LIN {X 0,Y 473.867,Z 372.012,A -85,B 0,C 180,E1 -7419.027,E2 -7419.027} C_VEL
LIN {X 0,Y 473.751,Z 376.078,A -85,B 0,C 180,E1 -7420.747,E2 -7420.747} C_VEL
LIN {X 0,Y 473.643,Z 378.041,A -85,B 0,C 180,E1 -7422.107,E2 -7422.107} C_VEL
LIN {X 0,Y 473.594,Z 378.94,A -85,B 0,C 180,E1 -7423.354,E2 -7423.354} C_VEL
LIN {X 0,Y 473.663,Z 378.958,A -85,B 0,C 180,E1 -7424.587,E2 -7424.587} C_VEL
LIN {X 0,Y 473.668,Z 378.173,A -85,B 0,C 180,E1 -7425.786,E2 -7425.786} C_VEL
LIN {X 0,Y 473.687,Z 376.639,A -85,B 0,C 180,E1 -7426.962,E2 -7426.962} C_VEL
LIN {X 0,Y 473.768,Z 374.355,A -85,B 0,C 180,E1 -7428.123,E2 -7428.123} C_VEL
LIN {X 0,Y 473.919,Z 369.986,A -85,B 0,C 180,E1 -7429.66,E2 -7429.66} C_VEL
LIN {X 0,Y 474.11,Z 365.022,A -85,B 0,C 180,E1 -7430.975,E2 -7430.975} C_VEL
LIN {X 0,Y 474.333,Z 358.198,A -85,B 0,C 180,E1 -7432.389,E2 -7432.389} C_VEL
LIN {X 0,Y 474.456,Z 355.246,A -85,B 0,C 180,E1 -7432.903,E2 -7432.903} C_VEL
LIN {X 0,Y 473.946,Z 351.766,A -85,B 0,C 180,E1 -7433.474,E2 -7433.474} C_VEL
LIN {X 0,Y 471.408,Z 345.796,A -85,B 0,C 180,E1 -7434.387,E2 -7434.387} C_VEL
LIN {X 0,Y 468.889,Z 339.334,A -85,B 0,C 180,E1 -7435.251,E2 -7435.251} C_VEL
LIN {X 0,Y 468.41,Z 335.005,A -85,B 0,C 180,E1 -7435.739,E2 -7435.739} C_VEL
LIN {X 0,Y 468.871,Z 324.63,A -85,B 0,C 180,E1 -7436.713,E2 -7436.713} C_VEL
LIN {X 0,Y 469.311,Z 314.156,A -85,B 0,C 180,E1 -7437.505,E2 -7437.505} C_VEL
LIN {X 0,Y 469.802,Z 301.748,A -85,B 0,C 180,E1 -7438.239,E2 -7438.239} C_VEL
LIN {X 0,Y 470.133,Z 288.339,A -85,B 0,C 180,E1 -7438.813,E2 -7438.813} C_VEL
LIN {X 0,Y 470.416,Z 274.959,A -85,B 0,C 180,E1 -7439.193,E2 -7439.193} C_VEL
LIN {X 0,Y 471.25,Z 183.279,A -85,B 0,C 180,E1 -7440.659,E2 -7440.659} C_VEL
LIN {X 0,Y 468.411,Z 168.295,A -85,B 0,C 180,E1 -7441.031,E2 -7441.031} C_VEL
LIN {X 0,Y 468.965,Z 153.603,A -85,B 0,C 180,E1 -7444.048,E2 -7444.048} C_VEL
LIN {X 0,Y 467.574,Z 145.244,A -85,B 0,C 180,E1 -7445.881,E2 -7445.881} C_VEL
LIN {X 0,Y 467.606,Z 145.236,A -85,B 0,C 180,E1 -7449.777,E2 -7449.777} C_VEL
LIN {X 0,Y 467.56,Z 145.247,A -85,B 0,C 180,E1 -7452.505,E2 -7452.505} C_VEL
LIN {X 0,Y 467.586,Z 145.236,A -85,B 0,C 180,E1 -7455.196,E2 -7455.196} C_VEL
LIN {X 0,Y 467.644,Z 145.231,A -85,B 0,C 180,E1 -7457.855,E2 -7457.855} C_VEL
LIN {X 0,Y 467.629,Z 145.231,A -85,B 0,C 180,E1 -7461.357,E2 -7461.357} C_VEL
LIN {X 0,Y 467.696,Z 145.227,A -85,B 0,C 180,E1 -7463.962,E2 -7463.962} C_VEL
LIN {X 0,Y 467.808,Z 145.209,A -85,B 0,C 180,E1 -7467.417,E2 -7467.417} C_VEL
LIN {X 0,Y 467.845,Z 145.211,A -85,B 0,C 180,E1 -7470,E2 -7470} C_VEL
LIN {X 0,Y 467.808,Z 145.21,A -85,B 0,C 180,E1 -7472.583,E2 -7472.583} C_VEL
LIN {X 0,Y 467.696,Z 145.229,A -85,B 0,C 180,E1 -7476.038,E2 -7476.038} C_VEL
LIN {X 0,Y 467.629,Z 145.231,A -85,B 0,C 180,E1 -7478.644,E2 -7478.644} C_VEL
LIN {X 0,Y 467.644,Z 145.232,A -85,B 0,C 180,E1 -7482.146,E2 -7482.146} C_VEL
LIN {X 0,Y 467.609,Z 145.241,A -85,B 0,C 180,E1 -7485.696,E2 -7485.696} C_VEL
LIN {X 0,Y 467.568,Z 145.238,A -85,B 0,C 180,E1 -7488.748,E2 -7488.748} C_VEL
LIN {X 0,Y 467.554,Z 145.243,A -85,B 0,C 180,E1 -7491.261,E2 -7491.261} C_VEL
LIN {X 0,Y 467.546,Z 145.244,A -85,B 0,C 180,E1 -7493.944,E2 -7493.944} C_VEL
LIN {X 0,Y 467.53,Z 145.244,A -85,B 0,C 180,E1 -7496.805,E2 -7496.805} C_VEL
LIN {X 0,Y 467.509,Z 145.249,A -85,B 0,C 180,E1 -7499.741,E2 -7499.741} C_VEL
LIN {X 0,Y 467.568,Z 145.239,A -85,B 0,C 180,E1 -7502.759,E2 -7502.759} C_VEL
LIN {X 0,Y 467.544,Z 145.242,A -85,B 0,C 180,E1 -7505.89,E2 -7505.89} C_VEL
LIN {X 0,Y 467.539,Z 145.249,A -85,B 0,C 180,E1 -7509.148,E2 -7509.148} C_VEL
LIN {X 0,Y 467.552,Z 145.245,A -85,B 0,C 180,E1 -7511.405,E2 -7511.405} C_VEL
LIN {X 0,Y 467.56,Z 145.247,A -85,B 0,C 180,E1 -7515.052,E2 -7515.052} C_VEL
LIN {X 0,Y 467.554,Z 145.244,A -85,B 0,C 180,E1 -7518.726,E2 -7518.726} C_VEL
LIN {X 0,Y 467.534,Z 145.242,A -85,B 0,C 180,E1 -7521.953,E2 -7521.953} C_VEL
LIN {X 0,Y 467.544,Z 145.245,A -85,B 0,C 180,E1 -7525.166,E2 -7525.166} C_VEL
LIN {X 0,Y 467.55,Z 145.242,A -85,B 0,C 180,E1 -7528.258,E2 -7528.258} C_VEL
LIN {X 0,Y 467.532,Z 145.244,A -85,B 0,C 180,E1 -7531.248,E2 -7531.248} C_VEL
LIN {X 0,Y 467.571,Z 145.243,A -85,B 0,C 180,E1 -7534.401,E2 -7534.401} C_VEL
LIN {X 0,Y 467.544,Z 145.244,A -85,B 0,C 180,E1 -7536.995,E2 -7536.995} C_VEL
LIN {X 0,Y 467.6,Z 145.235,A -85,B 0,C 180,E1 -7539.777,E2 -7539.777} C_VEL
LIN {X 0,Y 467.558,Z 145.247,A -85,B 0,C 180,E1 -7542.505,E2 -7542.505} C_VEL
LIN {X 0,Y 467.584,Z 145.237,A -85,B 0,C 180,E1 -7545.196,E2 -7545.196} C_VEL
LIN {X 0,Y 467.641,Z 145.231,A -85,B 0,C 180,E1 -7547.855,E2 -7547.855} C_VEL
LIN {X 0,Y 467.623,Z 145.231,A -85,B 0,C 180,E1 -7551.357,E2 -7551.357} C_VEL
LIN {X 0,Y 467.693,Z 145.227,A -85,B 0,C 180,E1 -7553.962,E2 -7553.962} C_VEL
LIN {X 0,Y 467.805,Z 145.209,A -85,B 0,C 180,E1 -7557.417,E2 -7557.417} C_VEL
LIN {X 0,Y 467.842,Z 145.211,A -85,B 0,C 180,E1 -7560,E2 -7560} C_VEL
LIN {X 0,Y 467.805,Z 145.21,A -85,B 0,C 180,E1 -7562.584,E2 -7562.584} C_VEL
LIN {X 0,Y 467.693,Z 145.229,A -85,B 0,C 180,E1 -7566.038,E2 -7566.038} C_VEL
LIN {X 0,Y 467.627,Z 145.231,A -85,B 0,C 180,E1 -7568.644,E2 -7568.644} C_VEL
LIN {X 0,Y 467.642,Z 145.232,A -85,B 0,C 180,E1 -7572.146,E2 -7572.146} C_VEL
LIN {X 0,Y 467.607,Z 145.241,A -85,B 0,C 180,E1 -7575.696,E2 -7575.696} C_VEL
LIN {X 0,Y 467.567,Z 145.238,A -85,B 0,C 180,E1 -7578.748,E2 -7578.748} C_VEL
LIN {X 0,Y 467.553,Z 145.244,A -85,B 0,C 180,E1 -7581.261,E2 -7581.261} C_VEL
LIN {X 0,Y 467.546,Z 145.244,A -85,B 0,C 180,E1 -7583.945,E2 -7583.945} C_VEL
LIN {X 0,Y 467.53,Z 145.244,A -85,B 0,C 180,E1 -7586.806,E2 -7586.806} C_VEL
LIN {X 0,Y 467.505,Z 145.249,A -85,B 0,C 180,E1 -7589.742,E2 -7589.742} C_VEL
LIN {X 0,Y 467.569,Z 145.24,A -85,B 0,C 180,E1 -7592.76,E2 -7592.76} C_VEL
LIN {X 0,Y 467.54,Z 145.243,A -85,B 0,C 180,E1 -7595.891,E2 -7595.891} C_VEL
LIN {X 0,Y 467.54,Z 145.25,A -85,B 0,C 180,E1 -7599.149,E2 -7599.149} C_VEL
LIN {X 0,Y 467.556,Z 145.244,A -85,B 0,C 180,E1 -7601.406,E2 -7601.406} C_VEL
LIN {X 0,Y 467.56,Z 145.247,A -85,B 0,C 180,E1 -7605.052,E2 -7605.052} C_VEL
LIN {X 0,Y 467.559,Z 145.244,A -85,B 0,C 180,E1 -7608.726,E2 -7608.726} C_VEL
LIN {X 0,Y 467.539,Z 145.242,A -85,B 0,C 180,E1 -7611.953,E2 -7611.953} C_VEL
LIN {X 0,Y 467.549,Z 145.244,A -85,B 0,C 180,E1 -7615.166,E2 -7615.166} C_VEL
LIN {X 0,Y 467.546,Z 145.243,A -85,B 0,C 180,E1 -7618.257,E2 -7618.257} C_VEL
LIN {X 0,Y 467.524,Z 145.247,A -85,B 0,C 180,E1 -7621.247,E2 -7621.247} C_VEL
LIN {X 0,Y 467.556,Z 145.305,A -85,B 0,C 180,E1 -7624.376,E2 -7624.376} C_VEL
LIN {X 0,Y 469.555,Z 155.653,A -85,B 0,C 180,E1 -7626.398,E2 -7626.398} C_VEL
LIN {X 0,Y 469.662,Z 160.735,A -85,B 0,C 180,E1 -7627.336,E2 -7627.336} C_VEL
LIN {X 0,Y 468.796,Z 180.844,A -85,B 0,C 180,E1 -7630.944,E2 -7630.944} C_VEL
LIN {X 0,Y 468.312,Z 192.554,A -85,B 0,C 180,E1 -7633.016,E2 -7633.016} C_VEL
LIN {X 0,Y 471.118,Z 211.466,A -85,B 0,C 180,E1 -7633.427,E2 -7633.427} C_VEL
LIN {X 0,Y 470.386,Z 301.176,A -85,B 0,C 180,E1 -7634.871,E2 -7634.871} C_VEL
LIN {X 0,Y 470.014,Z 314.178,A -85,B 0,C 180,E1 -7635.246,E2 -7635.246} C_VEL
LIN {X 0,Y 469.599,Z 326.238,A -85,B 0,C 180,E1 -7635.759,E2 -7635.759} C_VEL
LIN {X 0,Y 469.091,Z 338.452,A -85,B 0,C 180,E1 -7636.462,E2 -7636.462} C_VEL
LIN {X 0,Y 468.604,Z 349.481,A -85,B 0,C 180,E1 -7637.282,E2 -7637.282} C_VEL
LIN {X 0,Y 468.158,Z 360.491,A -85,B 0,C 180,E1 -7638.307,E2 -7638.307} C_VEL
LIN {X 0,Y 467.699,Z 369.878,A -85,B 0,C 180,E1 -7639.393,E2 -7639.393} C_VEL
LIN {X 0,Y 467.276,Z 378.958,A -85,B 0,C 180,E1 -7640.695,E2 -7640.695} C_VEL
LIN {X 0,Y 467.007,Z 386.273,A -85,B 0,C 180,E1 -7641.998,E2 -7641.998} C_VEL
LIN {X 0,Y 466.842,Z 391.213,A -85,B 0,C 180,E1 -7643.083,E2 -7643.083} C_VEL
LIN {X 0,Y 466.756,Z 396.008,A -85,B 0,C 180,E1 -7644.383,E2 -7644.383} C_VEL
LIN {X 0,Y 466.645,Z 399.671,A -85,B 0,C 180,E1 -7645.681,E2 -7645.681} C_VEL
LIN {X 0,Y 466.689,Z 401.563,A -85,B 0,C 180,E1 -7646.546,E2 -7646.546} C_VEL
LIN {X 0,Y 466.662,Z 402.984,A -85,B 0,C 180,E1 -7647.41,E2 -7647.41} C_VEL
LIN {X 0,Y 466.62,Z 404.604,A -85,B 0,C 180,E1 -7649.137,E2 -7649.137} C_VEL
LIN {X 0,Y 466.602,Z 404.824,A -85,B 0,C 180,E1 -7650,E2 -7650} C_VEL
LIN {X 0,Y 466.62,Z 404.606,A -85,B 0,C 180,E1 -7650.863,E2 -7650.863} C_VEL
LIN {X 0,Y 466.662,Z 402.978,A -85,B 0,C 180,E1 -7652.589,E2 -7652.589} C_VEL
LIN {X 0,Y 466.688,Z 401.562,A -85,B 0,C 180,E1 -7653.453,E2 -7653.453} C_VEL
LIN {X 0,Y 466.687,Z 398.586,A -85,B 0,C 180,E1 -7654.751,E2 -7654.751} C_VEL
LIN {X 0,Y 466.743,Z 394.561,A -85,B 0,C 180,E1 -7656.05,E2 -7656.05} C_VEL
LIN {X 0,Y 466.94,Z 388.369,A -85,B 0,C 180,E1 -7657.567,E2 -7657.567} C_VEL
LIN {X 0,Y 467.196,Z 381.607,A -85,B 0,C 180,E1 -7658.87,E2 -7658.87} C_VEL
LIN {X 0,Y 467.524,Z 373.225,A -85,B 0,C 180,E1 -7660.173,E2 -7660.173} C_VEL
LIN {X 0,Y 467.975,Z 364.611,A -85,B 0,C 180,E1 -7661.258,E2 -7661.258} C_VEL
LIN {X 0,Y 468.453,Z 354.527,A -85,B 0,C 180,E1 -7662.294,E2 -7662.294} C_VEL
LIN {X 0,Y 468.873,Z 343.464,A -85,B 0,C 180,E1 -7663.213,E2 -7663.213} C_VEL
LIN {X 0,Y 469.446,Z 331.882,A -85,B 0,C 180,E1 -7663.969,E2 -7663.969} C_VEL
LIN {X 0,Y 469.855,Z 319.883,A -85,B 0,C 180,E1 -7664.565,E2 -7664.565} C_VEL
LIN {X 0,Y 470.286,Z 306.964,A -85,B 0,C 180,E1 -7665.021,E2 -7665.021} C_VEL
LIN {X 0,Y 470.57,Z 293.349,A -85,B 0,C 180,E1 -7665.317,E2 -7665.317} C_VEL
LIN {X 0,Y 471.196,Z 210.389,A -85,B 0,C 180,E1 -7666.646,E2 -7666.646} C_VEL
LIN {X 0,Y 468.312,Z 191.835,A -85,B 0,C 180,E1 -7667.087,E2 -7667.087} C_VEL
LIN {X 0,Y 469.027,Z 174.329,A -85,B 0,C 180,E1 -7670.159,E2 -7670.159} C_VEL
LIN {X 0,Y 469.706,Z 157.643,A -85,B 0,C 180,E1 -7673.126,E2 -7673.126} C_VEL
LIN {X 0,Y 469.008,Z 152.49,A -85,B 0,C 180,E1 -7674.099,E2 -7674.099} C_VEL
LIN {X 0,Y 467.555,Z 145.247,A -85,B 0,C 180,E1 -7675.543,E2 -7675.543} C_VEL
LIN {X 0,Y 467.523,Z 145.251,A -85,B 0,C 180,E1 -7678.753,E2 -7678.753} C_VEL
LIN {X 0,Y 467.545,Z 145.249,A -85,B 0,C 180,E1 -7681.742,E2 -7681.742} C_VEL
LIN {X 0,Y 467.548,Z 145.246,A -85,B 0,C 180,E1 -7684.833,E2 -7684.833} C_VEL
LIN {X 0,Y 467.537,Z 145.245,A -85,B 0,C 180,E1 -7688.046,E2 -7688.046} C_VEL
LIN {X 0,Y 467.557,Z 145.248,A -85,B 0,C 180,E1 -7691.273,E2 -7691.273} C_VEL
LIN {X 0,Y 467.56,Z 145.246,A -85,B 0,C 180,E1 -7694.947,E2 -7694.947} C_VEL
LIN {X 0,Y 467.554,Z 145.244,A -85,B 0,C 180,E1 -7698.594,E2 -7698.594} C_VEL
LIN {X 0,Y 467.536,Z 145.245,A -85,B 0,C 180,E1 -7701.412,E2 -7701.412} C_VEL
LIN {X 0,Y 467.545,Z 145.242,A -85,B 0,C 180,E1 -7704.262,E2 -7704.262} C_VEL
LIN {X 0,Y 467.566,Z 145.239,A -85,B 0,C 180,E1 -7707.322,E2 -7707.322} C_VEL
LIN {X 0,Y 467.52,Z 145.248,A -85,B 0,C 180,E1 -7710.677,E2 -7710.677} C_VEL
LIN {X 0,Y 467.528,Z 145.241,A -85,B 0,C 180,E1 -7713.194,E2 -7713.194} C_VEL
LIN {X 0,Y 467.544,Z 145.245,A -85,B 0,C 180,E1 -7716.055,E2 -7716.055} C_VEL
LIN {X 0,Y 467.579,Z 145.239,A -85,B 0,C 180,E1 -7719.775,E2 -7719.775} C_VEL
LIN {X 0,Y 467.55,Z 145.247,A -85,B 0,C 180,E1 -7722.504,E2 -7722.504} C_VEL
LIN {X 0,Y 467.58,Z 145.235,A -85,B 0,C 180,E1 -7725.195,E2 -7725.195} C_VEL
LIN {X 0,Y 467.64,Z 145.233,A -85,B 0,C 180,E1 -7727.854,E2 -7727.854} C_VEL
LIN {X 0,Y 467.625,Z 145.231,A -85,B 0,C 180,E1 -7731.356,E2 -7731.356} C_VEL
LIN {X 0,Y 467.691,Z 145.231,A -85,B 0,C 180,E1 -7733.962,E2 -7733.962} C_VEL
LIN {X 0,Y 467.803,Z 145.212,A -85,B 0,C 180,E1 -7737.416,E2 -7737.416} C_VEL
LIN {X 0,Y 467.84,Z 145.211,A -85,B 0,C 180,E1 -7740,E2 -7740} C_VEL
LIN {X 0,Y 467.803,Z 145.211,A -85,B 0,C 180,E1 -7742.583,E2 -7742.583} C_VEL
LIN {X 0,Y 467.691,Z 145.23,A -85,B 0,C 180,E1 -7746.038,E2 -7746.038} C_VEL
LIN {X 0,Y 467.624,Z 145.234,A -85,B 0,C 180,E1 -7748.643,E2 -7748.643} C_VEL
LIN {X 0,Y 467.639,Z 145.237,A -85,B 0,C 180,E1 -7752.145,E2 -7752.145} C_VEL
LIN {X 0,Y 467.603,Z 145.244,A -85,B 0,C 180,E1 -7755.696,E2 -7755.696} C_VEL
LIN {X 0,Y 467.607,Z 145.241,A -85,B 0,C 180,E1 -7759.308,E2 -7759.308} C_VEL
LIN {X 0,Y 467.602,Z 145.344,A -85,B 0,C 180,E1 -7762.361,E2 -7762.361} C_VEL
LIN {X 0,Y 468.924,Z 152.789,A -85,B 0,C 180,E1 -7763.905,E2 -7763.905} C_VEL
LIN {X 0,Y 468.551,Z 168.51,A -85,B 0,C 180,E1 -7766.983,E2 -7766.983} C_VEL
LIN {X 0,Y 471.425,Z 184.218,A -85,B 0,C 180,E1 -7767.375,E2 -7767.375} C_VEL
LIN {X 0,Y 470.514,Z 276.407,A -85,B 0,C 180,E1 -7768.873,E2 -7768.873} C_VEL
LIN {X 0,Y 470.217,Z 289.972,A -85,B 0,C 180,E1 -7769.276,E2 -7769.276} C_VEL
LIN {X 0,Y 469.877,Z 302.576,A -85,B 0,C 180,E1 -7769.831,E2 -7769.831} C_VEL
LIN {X 0,Y 469.456,Z 313.602,A -85,B 0,C 180,E1 -7770.482,E2 -7770.482} C_VEL
LIN {X 0,Y 468.956,Z 324.82,A -85,B 0,C 180,E1 -7771.327,E2 -7771.327} C_VEL
LIN {X 0,Y 468.447,Z 335.259,A -85,B 0,C 180,E1 -7772.308,E2 -7772.308} C_VEL
LIN {X 0,Y 468.084,Z 344.387,A -85,B 0,C 180,E1 -7773.368,E2 -7773.368} C_VEL
LIN {X 0,Y 467.588,Z 353.449,A -85,B 0,C 180,E1 -7774.672,E2 -7774.672} C_VEL
LIN {X 0,Y 467.28,Z 360.415,A -85,B 0,C 180,E1 -7775.913,E2 -7775.913} C_VEL
LIN {X 0,Y 467.005,Z 365.825,A -85,B 0,C 180,E1 -7777.1,E2 -7777.1} C_VEL
LIN {X 0,Y 466.871,Z 370.84,A -85,B 0,C 180,E1 -7778.486,E2 -7778.486} C_VEL
LIN {X 0,Y 466.709,Z 374.498,A -85,B 0,C 180,E1 -7779.828,E2 -7779.828} C_VEL
LIN {X 0,Y 466.594,Z 377.553,A -85,B 0,C 180,E1 -7781.509,E2 -7781.509} C_VEL
LIN {X 0,Y 466.519,Z 378.782,A -85,B 0,C 180,E1 -7782.68,E2 -7782.68} C_VEL
LIN {X 0,Y 466.527,Z 379.234,A -85,B 0,C 180,E1 -7783.865,E2 -7783.865} C_VEL
LIN {X 0,Y 466.575,Z 378.93,A -85,B 0,C 180,E1 -7785.069,E2 -7785.069} C_VEL
LIN {X 0,Y 466.581,Z 377.824,A -85,B 0,C 180,E1 -7786.303,E2 -7786.303} C_VEL
LIN {X 0,Y 466.637,Z 375.844,A -85,B 0,C 180,E1 -7787.56,E2 -7787.56} C_VEL
LIN {X 0,Y 466.765,Z 372.897,A -85,B 0,C 180,E1 -7788.836,E2 -7788.836} C_VEL
LIN {X 0,Y 466.958,Z 367.587,A -85,B 0,C 180,E1 -7790.474,E2 -7790.474} C_VEL
LIN {X 0,Y 467.184,Z 361.377,A -85,B 0,C 180,E1 -7791.92,E2 -7791.92} C_VEL
LIN {X 0,Y 467.494,Z 353.742,A -85,B 0,C 180,E1 -7793.304,E2 -7793.304} C_VEL
LIN {X 0,Y 467.852,Z 345.917,A -85,B 0,C 180,E1 -7794.452,E2 -7794.452} C_VEL
LIN {X 0,Y 468.368,Z 336.18,A -85,B 0,C 180,E1 -7795.617,E2 -7795.617} C_VEL
LIN {X 0,Y 468.41,Z 335.005,A -85,B 0,C 180,E1 -7795.739,E2 -7795.739} C_VEL
LIN {X 0,Y 467.924,Z 330.526,A -85,B 0,C 180,E1 -7796.206,E2 -7796.206} C_VEL
LIN {X 0,Y 465.403,Z 323.026,A -85,B 0,C 180,E1 -7796.947,E2 -7796.947} C_VEL
LIN {X 0,Y 462.943,Z 315.158,A -85,B 0,C 180,E1 -7797.622,E2 -7797.622} C_VEL
LIN {X 0,Y 462.543,Z 310.011,A -85,B 0,C 180,E1 -7797.977,E2 -7797.977} C_VEL
LIN {X 0,Y 463.019,Z 297.561,A -85,B 0,C 180,E1 -7798.652,E2 -7798.652} C_VEL
LIN {X 0,Y 463.349,Z 284.424,A -85,B 0,C 180,E1 -7799.159,E2 -7799.159} C_VEL
LIN {X 0,Y 463.563,Z 271.09,A -85,B 0,C 180,E1 -7799.484,E2 -7799.484} C_VEL
LIN {X 0,Y 464.339,Z 183.536,A -85,B 0,C 180,E1 -7800.899,E2 -7800.899} C_VEL
LIN {X 0,Y 461.446,Z 168.527,A -85,B 0,C 180,E1 -7801.269,E2 -7801.269} C_VEL
LIN {X 0,Y 461.998,Z 155.035,A -85,B 0,C 180,E1 -7804.076,E2 -7804.076} C_VEL
LIN {X 0,Y 460.548,Z 146.12,A -85,B 0,C 180,E1 -7806.064,E2 -7806.064} C_VEL
LIN {X 0,Y 460.534,Z 146.117,A -85,B 0,C 180,E1 -7809.452,E2 -7809.452} C_VEL
LIN {X 0,Y 460.519,Z 146.121,A -85,B 0,C 180,E1 -7812.229,E2 -7812.229} C_VEL
LIN {X 0,Y 460.544,Z 146.115,A -85,B 0,C 180,E1 -7814.965,E2 -7814.965} C_VEL
LIN {X 0,Y 460.588,Z 146.113,A -85,B 0,C 180,E1 -7818.559,E2 -7818.559} C_VEL
LIN {X 0,Y 460.619,Z 146.11,A -85,B 0,C 180,E1 -7822.107,E2 -7822.107} C_VEL
LIN {X 0,Y 460.668,Z 146.099,A -85,B 0,C 180,E1 -7824.748,E2 -7824.748} C_VEL
LIN {X 0,Y 460.752,Z 146.088,A -85,B 0,C 180,E1 -7827.377,E2 -7827.377} C_VEL
LIN {X 0,Y 460.815,Z 146.086,A -85,B 0,C 180,E1 -7830,E2 -7830} C_VEL
LIN {X 0,Y 460.751,Z 146.089,A -85,B 0,C 180,E1 -7832.623,E2 -7832.623} C_VEL
LIN {X 0,Y 460.662,Z 146.104,A -85,B 0,C 180,E1 -7836.131,E2 -7836.131} C_VEL
LIN {X 0,Y 460.584,Z 146.108,A -85,B 0,C 180,E1 -7838.777,E2 -7838.777} C_VEL
LIN {X 0,Y 460.594,Z 146.108,A -85,B 0,C 180,E1 -7842.435,E2 -7842.435} C_VEL
LIN {X 0,Y 460.554,Z 146.117,A -85,B 0,C 180,E1 -7845.978,E2 -7845.978} C_VEL
LIN {X 0,Y 460.526,Z 146.116,A -85,B 0,C 180,E1 -7848.886,E2 -7848.886} C_VEL
LIN {X 0,Y 460.505,Z 146.124,A -85,B 0,C 180,E1 -7851.486,E2 -7851.486} C_VEL
LIN {X 0,Y 460.51,Z 146.118,A -85,B 0,C 180,E1 -7854.334,E2 -7854.334} C_VEL
LIN {X 0,Y 460.484,Z 146.126,A -85,B 0,C 180,E1 -7857.249,E2 -7857.249} C_VEL
LIN {X 0,Y 460.478,Z 146.122,A -85,B 0,C 180,E1 -7860.242,E2 -7860.242} C_VEL
LIN {X 0,Y 460.511,Z 146.125,A -85,B 0,C 180,E1 -7863.326,E2 -7863.326} C_VEL
LIN {X 0,Y 460.464,Z 146.124,A -85,B 0,C 180,E1 -7866.53,E2 -7866.53} C_VEL
LIN {X 0,Y 460.505,Z 146.119,A -85,B 0,C 180,E1 -7869.865,E2 -7869.865} C_VEL
LIN {X 0,Y 460.456,Z 146.129,A -85,B 0,C 180,E1 -7872.893,E2 -7872.893} C_VEL
LIN {X 0,Y 460.497,Z 146.119,A -85,B 0,C 180,E1 -7875.832,E2 -7875.832} C_VEL
LIN {X 0,Y 460.508,Z 146.126,A -85,B 0,C 180,E1 -7878.987,E2 -7878.987} C_VEL
LIN {X 0,Y 460.477,Z 146.123,A -85,B 0,C 180,E1 -7882.375,E2 -7882.375} C_VEL
LIN {X 0,Y 460.527,Z 146.116,A -85,B 0,C 180,E1 -7885.623,E2 -7885.623} C_VEL
LIN {X 0,Y 460.498,Z 146.127,A -85,B 0,C 180,E1 -7888.742,E2 -7888.742} C_VEL
LIN {X 0,Y 460.497,Z 146.119,A -85,B 0,C 180,E1 -7891.764,E2 -7891.764} C_VEL
LIN {X 0,Y 460.515,Z 146.124,A -85,B 0,C 180,E1 -7894.703,E2 -7894.703} C_VEL
LIN {X 0,Y 460.489,Z 146.12,A -85,B 0,C 180,E1 -7897.571,E2 -7897.571} C_VEL
LIN {X 0,Y 460.553,Z 146.118,A -85,B 0,C 180,E1 -7900.384,E2 -7900.384} C_VEL
LIN {X 0,Y 460.56,Z 146.114,A -85,B 0,C 180,E1 -7904.058,E2 -7904.058} C_VEL
LIN {X 0,Y 460.596,Z 146.107,A -85,B 0,C 180,E1 -7907.666,E2 -7907.666} C_VEL
LIN {X 0,Y 460.578,Z 146.109,A -85,B 0,C 180,E1 -7911.223,E2 -7911.223} C_VEL
LIN {X 0,Y 460.659,Z 146.102,A -85,B 0,C 180,E1 -7913.87,E2 -7913.87} C_VEL
LIN {X 0,Y 460.749,Z 146.088,A -85,B 0,C 180,E1 -7917.378,E2 -7917.378} C_VEL
LIN {X 0,Y 460.812,Z 146.087,A -85,B 0,C 180,E1 -7920,E2 -7920} C_VEL
LIN {X 0,Y 460.749,Z 146.089,A -85,B 0,C 180,E1 -7922.623,E2 -7922.623} C_VEL
LIN {X 0,Y 460.66,Z 146.104,A -85,B 0,C 180,E1 -7926.131,E2 -7926.131} C_VEL
LIN {X 0,Y 460.582,Z 146.108,A -85,B 0,C 180,E1 -7928.777,E2 -7928.777} C_VEL
LIN {X 0,Y 460.592,Z 146.108,A -85,B 0,C 180,E1 -7932.435,E2 -7932.435} C_VEL
LIN {X 0,Y 460.552,Z 146.116,A -85,B 0,C 180,E1 -7935.979,E2 -7935.979} C_VEL
LIN {X 0,Y 460.525,Z 146.116,A -85,B 0,C 180,E1 -7938.887,E2 -7938.887} C_VEL
LIN {X 0,Y 460.504,Z 146.125,A -85,B 0,C 180,E1 -7941.487,E2 -7941.487} C_VEL
LIN {X 0,Y 460.51,Z 146.118,A -85,B 0,C 180,E1 -7944.334,E2 -7944.334} C_VEL
LIN {X 0,Y 460.485,Z 146.126,A -85,B 0,C 180,E1 -7947.25,E2 -7947.25} C_VEL
LIN {X 0,Y 460.474,Z 146.122,A -85,B 0,C 180,E1 -7950.243,E2 -7950.243} C_VEL
LIN {X 0,Y 460.512,Z 146.125,A -85,B 0,C 180,E1 -7953.327,E2 -7953.327} C_VEL
LIN {X 0,Y 460.457,Z 146.125,A -85,B 0,C 180,E1 -7956.532,E2 -7956.532} C_VEL
LIN {X 0,Y 460.507,Z 146.119,A -85,B 0,C 180,E1 -7959.865,E2 -7959.865} C_VEL
LIN {X 0,Y 460.454,Z 146.13,A -85,B 0,C 180,E1 -7962.893,E2 -7962.893} C_VEL
LIN {X 0,Y 460.502,Z 146.119,A -85,B 0,C 180,E1 -7965.832,E2 -7965.832} C_VEL
LIN {X 0,Y 460.513,Z 146.125,A -85,B 0,C 180,E1 -7968.987,E2 -7968.987} C_VEL
LIN {X 0,Y 460.481,Z 146.123,A -85,B 0,C 180,E1 -7972.375,E2 -7972.375} C_VEL
LIN {X 0,Y 460.533,Z 146.115,A -85,B 0,C 180,E1 -7975.623,E2 -7975.623} C_VEL
LIN {X 0,Y 460.504,Z 146.126,A -85,B 0,C 180,E1 -7978.742,E2 -7978.742} C_VEL
LIN {X 0,Y 460.495,Z 146.121,A -85,B 0,C 180,E1 -7981.764,E2 -7981.764} C_VEL
LIN {X 0,Y 460.54,Z 146.131,A -85,B 0,C 180,E1 -7984.164,E2 -7984.164} C_VEL
LIN {X 0,Y 462.716,Z 157.95,A -85,B 0,C 180,E1 -7986.503,E2 -7986.503} C_VEL
LIN {X 0,Y 462.441,Z 167.575,A -85,B 0,C 180,E1 -7988.279,E2 -7988.279} C_VEL
LIN {X 0,Y 461.645,Z 184.547,A -85,B 0,C 180,E1 -7991.355,E2 -7991.355} C_VEL
LIN {X 0,Y 461.338,Z 192.334,A -85,B 0,C 180,E1 -7992.755,E2 -7992.755} C_VEL
LIN {X 0,Y 464.288,Z 211.601,A -85,B 0,C 180,E1 -7993.192,E2 -7993.192} C_VEL
LIN {X 0,Y 463.491,Z 300.335,A -85,B 0,C 180,E1 -7994.64,E2 -7994.64} C_VEL
LIN {X 0,Y 463.138,Z 313.551,A -85,B 0,C 180,E1 -7995.022,E2 -7995.022} C_VEL
LIN {X 0,Y 462.7,Z 325.723,A -85,B 0,C 180,E1 -7995.542,E2 -7995.542} C_VEL
LIN {X 0,Y 462.161,Z 338.038,A -85,B 0,C 180,E1 -7996.255,E2 -7996.255} C_VEL
LIN {X 0,Y 461.598,Z 350.128,A -85,B 0,C 180,E1 -7997.173,E2 -7997.173} C_VEL
LIN {X 0,Y 461.107,Z 361.204,A -85,B 0,C 180,E1 -7998.237,E2 -7998.237} C_VEL
LIN {X 0,Y 460.562,Z 371.224,A -85,B 0,C 180,E1 -7999.449,E2 -7999.449} C_VEL
LIN {X 0,Y 460.183,Z 380.051,A -85,B 0,C 180,E1 -8000.772,E2 -8000.772} C_VEL
LIN {X 0,Y 459.889,Z 387.085,A -85,B 0,C 180,E1 -8002.095,E2 -8002.095} C_VEL
LIN {X 0,Y 459.693,Z 393.367,A -85,B 0,C 180,E1 -8003.593,E2 -8003.593} C_VEL
LIN {X 0,Y 459.615,Z 398.372,A -85,B 0,C 180,E1 -8005.176,E2 -8005.176} C_VEL
LIN {X 0,Y 459.583,Z 401.351,A -85,B 0,C 180,E1 -8006.493,E2 -8006.493} C_VEL
LIN {X 0,Y 459.585,Z 402.779,A -85,B 0,C 180,E1 -8007.37,E2 -8007.37} C_VEL
LIN {X 0,Y 459.523,Z 404.405,A -85,B 0,C 180,E1 -8009.124,E2 -8009.124} C_VEL
LIN {X 0,Y 459.533,Z 404.629,A -85,B 0,C 180,E1 -8010,E2 -8010} C_VEL
LIN {X 0,Y 459.523,Z 404.414,A -85,B 0,C 180,E1 -8010.876,E2 -8010.876} C_VEL
LIN {X 0,Y 459.584,Z 402.788,A -85,B 0,C 180,E1 -8012.629,E2 -8012.629} C_VEL
LIN {X 0,Y 459.583,Z 401.373,A -85,B 0,C 180,E1 -8013.507,E2 -8013.507} C_VEL
LIN {X 0,Y 459.615,Z 398.399,A -85,B 0,C 180,E1 -8014.824,E2 -8014.824} C_VEL
LIN {X 0,Y 459.715,Z 393.331,A -85,B 0,C 180,E1 -8016.431,E2 -8016.431} C_VEL
LIN {X 0,Y 459.898,Z 387.165,A -85,B 0,C 180,E1 -8017.905,E2 -8017.905} C_VEL
LIN {X 0,Y 460.19,Z 380.181,A -85,B 0,C 180,E1 -8019.227,E2 -8019.227} C_VEL
LIN {X 0,Y 460.504,Z 373.05,A -85,B 0,C 180,E1 -8020.33,E2 -8020.33} C_VEL
LIN {X 0,Y 460.983,Z 364.44,A -85,B 0,C 180,E1 -8021.431,E2 -8021.431} C_VEL
LIN {X 0,Y 461.49,Z 354.557,A -85,B 0,C 180,E1 -8022.463,E2 -8022.463} C_VEL
LIN {X 0,Y 461.941,Z 343.31,A -85,B 0,C 180,E1 -8023.415,E2 -8023.415} C_VEL
LIN {X 0,Y 462.539,Z 331.757,A -85,B 0,C 180,E1 -8024.182,E2 -8024.182} C_VEL
LIN {X 0,Y 462.991,Z 319.801,A -85,B 0,C 180,E1 -8024.785,E2 -8024.785} C_VEL
LIN {X 0,Y 463.503,Z 306.05,A -85,B 0,C 180,E1 -8025.275,E2 -8025.275} C_VEL
LIN {X 0,Y 463.732,Z 293.569,A -85,B 0,C 180,E1 -8025.548,E2 -8025.548} C_VEL
LIN {X 0,Y 464.394,Z 210.91,A -85,B 0,C 180,E1 -8026.897,E2 -8026.897} C_VEL
LIN {X 0,Y 461.35,Z 191.663,A -85,B 0,C 180,E1 -8027.361,E2 -8027.361} C_VEL
LIN {X 0,Y 462.077,Z 174.191,A -85,B 0,C 180,E1 -8030.476,E2 -8030.476} C_VEL
LIN {X 0,Y 462.779,Z 158.816,A -85,B 0,C 180,E1 -8033.256,E2 -8033.256} C_VEL
LIN {X 0,Y 461.804,Z 152.369,A -85,B 0,C 180,E1 -8034.5,E2 -8034.5} C_VEL
LIN {X 0,Y 460.521,Z 146.123,A -85,B 0,C 180,E1 -8035.789,E2 -8035.789} C_VEL
LIN {X 0,Y 460.494,Z 146.126,A -85,B 0,C 180,E1 -8038.236,E2 -8038.236} C_VEL
LIN {X 0,Y 460.494,Z 146.13,A -85,B 0,C 180,E1 -8041.277,E2 -8041.277} C_VEL
LIN {X 0,Y 460.517,Z 146.12,A -85,B 0,C 180,E1 -8044.502,E2 -8044.502} C_VEL
LIN {X 0,Y 460.48,Z 146.127,A -85,B 0,C 180,E1 -8047.624,E2 -8047.624} C_VEL
LIN {X 0,Y 460.511,Z 146.126,A -85,B 0,C 180,E1 -8051.012,E2 -8051.012} C_VEL
LIN {X 0,Y 460.507,Z 146.125,A -85,B 0,C 180,E1 -8054.589,E2 -8054.589} C_VEL
LIN {X 0,Y 460.469,Z 146.122,A -85,B 0,C 180,E1 -8057.812,E2 -8057.812} C_VEL
LIN {X 0,Y 460.505,Z 146.119,A -85,B 0,C 180,E1 -8060.134,E2 -8060.134} C_VEL
LIN {X 0,Y 460.455,Z 146.123,A -85,B 0,C 180,E1 -8063.468,E2 -8063.468} C_VEL
LIN {X 0,Y 460.511,Z 146.12,A -85,B 0,C 180,E1 -8066.673,E2 -8066.673} C_VEL
LIN {X 0,Y 460.472,Z 146.121,A -85,B 0,C 180,E1 -8069.757,E2 -8069.757} C_VEL
LIN {X 0,Y 460.482,Z 146.123,A -85,B 0,C 180,E1 -8072.75,E2 -8072.75} C_VEL
LIN {X 0,Y 460.508,Z 146.119,A -85,B 0,C 180,E1 -8075.665,E2 -8075.665} C_VEL
LIN {X 0,Y 460.507,Z 146.125,A -85,B 0,C 180,E1 -8078.58,E2 -8078.58} C_VEL
LIN {X 0,Y 460.523,Z 146.113,A -85,B 0,C 180,E1 -8081.308,E2 -8081.308} C_VEL
LIN {X 0,Y 460.56,Z 146.117,A -85,B 0,C 180,E1 -8084.057,E2 -8084.057} C_VEL
LIN {X 0,Y 460.596,Z 146.109,A -85,B 0,C 180,E1 -8087.665,E2 -8087.665} C_VEL
LIN {X 0,Y 460.58,Z 146.109,A -85,B 0,C 180,E1 -8091.223,E2 -8091.223} C_VEL
LIN {X 0,Y 460.658,Z 146.105,A -85,B 0,C 180,E1 -8093.869,E2 -8093.869} C_VEL
LIN {X 0,Y 460.747,Z 146.091,A -85,B 0,C 180,E1 -8097.377,E2 -8097.377} C_VEL
LIN {X 0,Y 460.81,Z 146.086,A -85,B 0,C 180,E1 -8100,E2 -8100} C_VEL
LIN {X 0,Y 460.747,Z 146.09,A -85,B 0,C 180,E1 -8102.622,E2 -8102.622} C_VEL
LIN {X 0,Y 460.657,Z 146.105,A -85,B 0,C 180,E1 -8106.13,E2 -8106.13} C_VEL
LIN {X 0,Y 460.579,Z 146.112,A -85,B 0,C 180,E1 -8108.777,E2 -8108.777} C_VEL
LIN {X 0,Y 460.589,Z 146.114,A -85,B 0,C 180,E1 -8112.435,E2 -8112.435} C_VEL
LIN {X 0,Y 460.549,Z 146.121,A -85,B 0,C 180,E1 -8115.978,E2 -8115.978} C_VEL
LIN {X 0,Y 460.552,Z 146.121,A -85,B 0,C 180,E1 -8119.616,E2 -8119.616} C_VEL
LIN {X 0,Y 460.546,Z 146.173,A -85,B 0,C 180,E1 -8122.131,E2 -8122.131} C_VEL
LIN {X 0,Y 461.936,Z 153.642,A -85,B 0,C 180,E1 -8123.711,E2 -8123.711} C_VEL
LIN {X 0,Y 461.664,Z 167.375,A -85,B 0,C 180,E1 -8126.441,E2 -8126.441} C_VEL
LIN {X 0,Y 461.607,Z 168.807,A -85,B 0,C 180,E1 -8126.719,E2 -8126.719} C_VEL
LIN {X 0,Y 464.64,Z 184.235,A -85,B 0,C 180,E1 -8127.107,E2 -8127.107} C_VEL
LIN {X 0,Y 463.693,Z 276.755,A -85,B 0,C 180,E1 -8128.641,E2 -8128.641} C_VEL
LIN {X 0,Y 463.361,Z 289.902,A -85,B 0,C 180,E1 -8129.035,E2 -8129.035} C_VEL
LIN {X 0,Y 463.007,Z 302.985,A -85,B 0,C 180,E1 -8129.621,E2 -8129.621} C_VEL
LIN {X 0,Y 462.513,Z 314.898,A -85,B 0,C 180,E1 -8130.347,E2 -8130.347} C_VEL
LIN {X 0,Y 461.966,Z 326.368,A -85,B 0,C 180,E1 -8131.243,E2 -8131.243} C_VEL
LIN {X 0,Y 461.466,Z 336.282,A -85,B 0,C 180,E1 -8132.211,E2 -8132.211} C_VEL
LIN {X 0,Y 460.975,Z 346.21,A -85,B 0,C 180,E1 -8133.419,E2 -8133.419} C_VEL
LIN {X 0,Y 460.512,Z 354.69,A -85,B 0,C 180,E1 -8134.692,E2 -8134.692} C_VEL
LIN {X 0,Y 460.197,Z 361.528,A -85,B 0,C 180,E1 -8135.964,E2 -8135.964} C_VEL
LIN {X 0,Y 459.938,Z 367.581,A -85,B 0,C 180,E1 -8137.386,E2 -8137.386} C_VEL
LIN {X 0,Y 459.728,Z 372.268,A -85,B 0,C 180,E1 -8138.812,E2 -8138.812} C_VEL
LIN {X 0,Y 459.6,Z 375.495,A -85,B 0,C 180,E1 -8140.132,E2 -8140.132} C_VEL
LIN {X 0,Y 459.501,Z 377.745,A -85,B 0,C 180,E1 -8141.459,E2 -8141.459} C_VEL
LIN {X 0,Y 459.43,Z 379.036,A -85,B 0,C 180,E1 -8142.756,E2 -8142.756} C_VEL
LIN {X 0,Y 459.44,Z 379.452,A -85,B 0,C 180,E1 -8144.033,E2 -8144.033} C_VEL
LIN {X 0,Y 459.477,Z 379.007,A -85,B 0,C 180,E1 -8145.285,E2 -8145.285} C_VEL
LIN {X 0,Y 459.508,Z 377.783,A -85,B 0,C 180,E1 -8146.509,E2 -8146.509} C_VEL
LIN {X 0,Y 459.549,Z 375.819,A -85,B 0,C 180,E1 -8147.709,E2 -8147.709} C_VEL
LIN {X 0,Y 459.731,Z 371.656,A -85,B 0,C 180,E1 -8149.404,E2 -8149.404} C_VEL
LIN {X 0,Y 459.926,Z 366.386,A -85,B 0,C 180,E1 -8150.927,E2 -8150.927} C_VEL
LIN {X 0,Y 460.187,Z 359.961,A -85,B 0,C 180,E1 -8152.348,E2 -8152.348} C_VEL
LIN {X 0,Y 460.573,Z 351.959,A -85,B 0,C 180,E1 -8153.751,E2 -8153.751} C_VEL
LIN {X 0,Y 461.018,Z 342.921,A -85,B 0,C 180,E1 -8155.012,E2 -8155.012} C_VEL
LIN {X 0,Y 461.532,Z 333.254,A -85,B 0,C 180,E1 -8156.103,E2 -8156.103} C_VEL
LIN {X 0,Y 462.052,Z 322.807,A -85,B 0,C 180,E1 -8157.06,E2 -8157.06} C_VEL
LIN {X 0,Y 462.454,Z 311.789,A -85,B 0,C 180,E1 -8157.867,E2 -8157.867} C_VEL
LIN {X 0,Y 462.543,Z 310.011,A -85,B 0,C 180,E1 -8157.977,E2 -8157.977} C_VEL
LIN {X 0,Y 462.183,Z 304.752,A -85,B 0,C 180,E1 -8158.305,E2 -8158.305} C_VEL
LIN {X 0,Y 459.79,Z 296.078,A -85,B 0,C 180,E1 -8158.821,E2 -8158.821} C_VEL
LIN {X 0,Y 457.222,Z 287.18,A -85,B 0,C 180,E1 -8159.264,E2 -8159.264} C_VEL
LIN {X 0,Y 456.55,Z 281.545,A -85,B 0,C 180,E1 -8159.467,E2 -8159.467} C_VEL
LIN {X 0,Y 456.749,Z 267.243,A -85,B 0,C 180,E1 -8159.773,E2 -8159.773} C_VEL
LIN {X 0,Y 457.546,Z 184.602,A -85,B 0,C 180,E1 -8161.13,E2 -8161.13} C_VEL
LIN {X 0,Y 454.502,Z 168.724,A -85,B 0,C 180,E1 -8161.522,E2 -8161.522} C_VEL
LIN {X 0,Y 455.041,Z 156.916,A -85,B 0,C 180,E1 -8164.006,E2 -8164.006} C_VEL
LIN {X 0,Y 454.412,Z 152.086,A -85,B 0,C 180,E1 -8165.074,E2 -8165.074} C_VEL
LIN {X 0,Y 453.51,Z 146.996,A -85,B 0,C 180,E1 -8166.24,E2 -8166.24} C_VEL
LIN {X 0,Y 453.469,Z 146.998,A -85,B 0,C 180,E1 -8169.117,E2 -8169.117} C_VEL
LIN {X 0,Y 453.48,Z 146.995,A -85,B 0,C 180,E1 -8171.944,E2 -8171.944} C_VEL
LIN {X 0,Y 453.514,Z 146.993,A -85,B 0,C 180,E1 -8174.726,E2 -8174.726} C_VEL
LIN {X 0,Y 453.54,Z 146.993,A -85,B 0,C 180,E1 -8178.379,E2 -8178.379} C_VEL
LIN {X 0,Y 453.554,Z 146.984,A -85,B 0,C 180,E1 -8181.086,E2 -8181.086} C_VEL
LIN {X 0,Y 453.63,Z 146.977,A -85,B 0,C 180,E1 -8183.774,E2 -8183.774} C_VEL
LIN {X 0,Y 453.699,Z 146.966,A -85,B 0,C 180,E1 -8187.337,E2 -8187.337} C_VEL
LIN {X 0,Y 453.764,Z 146.965,A -85,B 0,C 180,E1 -8190,E2 -8190} C_VEL
LIN {X 0,Y 453.698,Z 146.967,A -85,B 0,C 180,E1 -8192.664,E2 -8192.664} C_VEL
LIN {X 0,Y 453.63,Z 146.979,A -85,B 0,C 180,E1 -8196.226,E2 -8196.226} C_VEL
LIN {X 0,Y 453.554,Z 146.984,A -85,B 0,C 180,E1 -8198.914,E2 -8198.914} C_VEL
LIN {X 0,Y 453.561,Z 146.984,A -85,B 0,C 180,E1 -8202.529,E2 -8202.529} C_VEL
LIN {X 0,Y 453.493,Z 146.994,A -85,B 0,C 180,E1 -8206.198,E2 -8206.198} C_VEL
LIN {X 0,Y 453.481,Z 146.994,A -85,B 0,C 180,E1 -8209.027,E2 -8209.027} C_VEL
LIN {X 0,Y 453.465,Z 147,A -85,B 0,C 180,E1 -8211.837,E2 -8211.837} C_VEL
LIN {X 0,Y 453.464,Z 146.995,A -85,B 0,C 180,E1 -8214.737,E2 -8214.737} C_VEL
LIN {X 0,Y 453.453,Z 146.999,A -85,B 0,C 180,E1 -8217.941,E2 -8217.941} C_VEL
LIN {X 0,Y 453.444,Z 146.999,A -85,B 0,C 180,E1 -8220.762,E2 -8220.762} C_VEL
LIN {X 0,Y 453.461,Z 146.997,A -85,B 0,C 180,E1 -8223.914,E2 -8223.914} C_VEL
LIN {X 0,Y 453.441,Z 147.005,A -85,B 0,C 180,E1 -8227.19,E2 -8227.19} C_VEL
LIN {X 0,Y 453.464,Z 146.997,A -85,B 0,C 180,E1 -8230.612,E2 -8230.612} C_VEL
LIN {X 0,Y 453.475,Z 146.995,A -85,B 0,C 180,E1 -8234.528,E2 -8234.528} C_VEL
LIN {X 0,Y 453.43,Z 146.999,A -85,B 0,C 180,E1 -8238.071,E2 -8238.071} C_VEL
LIN {X 0,Y 453.433,Z 147.005,A -85,B 0,C 180,E1 -8240.802,E2 -8240.802} C_VEL
LIN {X 0,Y 453.436,Z 146.999,A -85,B 0,C 180,E1 -8243.916,E2 -8243.916} C_VEL
LIN {X 0,Y 453.467,Z 146.998,A -85,B 0,C 180,E1 -8247.15,E2 -8247.15} C_VEL
LIN {X 0,Y 453.449,Z 146.999,A -85,B 0,C 180,E1 -8250.267,E2 -8250.267} C_VEL
LIN {X 0,Y 453.435,Z 147,A -85,B 0,C 180,E1 -8253.29,E2 -8253.29} C_VEL
LIN {X 0,Y 453.474,Z 146.997,A -85,B 0,C 180,E1 -8256.238,E2 -8256.238} C_VEL
LIN {X 0,Y 453.464,Z 146.996,A -85,B 0,C 180,E1 -8259.117,E2 -8259.117} C_VEL
LIN {X 0,Y 453.478,Z 146.995,A -85,B 0,C 180,E1 -8261.944,E2 -8261.944} C_VEL
LIN {X 0,Y 453.511,Z 146.993,A -85,B 0,C 180,E1 -8264.726,E2 -8264.726} C_VEL
LIN {X 0,Y 453.537,Z 146.993,A -85,B 0,C 180,E1 -8268.379,E2 -8268.379} C_VEL
LIN {X 0,Y 453.549,Z 146.985,A -85,B 0,C 180,E1 -8271.086,E2 -8271.086} C_VEL
LIN {X 0,Y 453.627,Z 146.977,A -85,B 0,C 180,E1 -8273.774,E2 -8273.774} C_VEL
LIN {X 0,Y 453.696,Z 146.967,A -85,B 0,C 180,E1 -8277.337,E2 -8277.337} C_VEL
LIN {X 0,Y 453.761,Z 146.965,A -85,B 0,C 180,E1 -8280,E2 -8280} C_VEL
LIN {X 0,Y 453.695,Z 146.967,A -85,B 0,C 180,E1 -8282.664,E2 -8282.664} C_VEL
LIN {X 0,Y 453.628,Z 146.979,A -85,B 0,C 180,E1 -8286.226,E2 -8286.226} C_VEL
LIN {X 0,Y 453.552,Z 146.984,A -85,B 0,C 180,E1 -8288.915,E2 -8288.915} C_VEL
LIN {X 0,Y 453.56,Z 146.984,A -85,B 0,C 180,E1 -8292.529,E2 -8292.529} C_VEL
LIN {X 0,Y 453.492,Z 146.994,A -85,B 0,C 180,E1 -8296.198,E2 -8296.198} C_VEL
LIN {X 0,Y 453.481,Z 146.994,A -85,B 0,C 180,E1 -8299.028,E2 -8299.028} C_VEL
LIN {X 0,Y 453.465,Z 146.999,A -85,B 0,C 180,E1 -8301.837,E2 -8301.837} C_VEL
LIN {X 0,Y 453.464,Z 146.996,A -85,B 0,C 180,E1 -8304.738,E2 -8304.738} C_VEL
LIN {X 0,Y 453.453,Z 146.998,A -85,B 0,C 180,E1 -8307.942,E2 -8307.942} C_VEL
LIN {X 0,Y 453.443,Z 146.999,A -85,B 0,C 180,E1 -8310.762,E2 -8310.762} C_VEL
LIN {X 0,Y 453.462,Z 146.997,A -85,B 0,C 180,E1 -8313.914,E2 -8313.914} C_VEL
LIN {X 0,Y 453.433,Z 147.007,A -85,B 0,C 180,E1 -8317.192,E2 -8317.192} C_VEL
LIN {X 0,Y 453.468,Z 146.996,A -85,B 0,C 180,E1 -8320.612,E2 -8320.612} C_VEL
LIN {X 0,Y 453.479,Z 146.995,A -85,B 0,C 180,E1 -8324.529,E2 -8324.529} C_VEL
LIN {X 0,Y 453.433,Z 146.999,A -85,B 0,C 180,E1 -8328.072,E2 -8328.072} C_VEL
LIN {X 0,Y 453.437,Z 147.005,A -85,B 0,C 180,E1 -8330.803,E2 -8330.803} C_VEL
LIN {X 0,Y 453.44,Z 146.998,A -85,B 0,C 180,E1 -8333.916,E2 -8333.916} C_VEL
LIN {X 0,Y 453.471,Z 146.999,A -85,B 0,C 180,E1 -8337.151,E2 -8337.151} C_VEL
LIN {X 0,Y 453.447,Z 147,A -85,B 0,C 180,E1 -8340.267,E2 -8340.267} C_VEL
LIN {X 0,Y 453.436,Z 147,A -85,B 0,C 180,E1 -8343.29,E2 -8343.29} C_VEL
LIN {X 0,Y 453.487,Z 147.123,A -85,B 0,C 180,E1 -8343.977,E2 -8343.977} C_VEL
LIN {X 0,Y 455.724,Z 158.964,A -85,B 0,C 180,E1 -8346.362,E2 -8346.362} C_VEL
LIN {X 0,Y 455.57,Z 167.09,A -85,B 0,C 180,E1 -8347.889,E2 -8347.889} C_VEL
LIN {X 0,Y 454.718,Z 184.294,A -85,B 0,C 180,E1 -8351.061,E2 -8351.061} C_VEL
LIN {X 0,Y 454.356,Z 192.225,A -85,B 0,C 180,E1 -8352.508,E2 -8352.508} C_VEL
LIN {X 0,Y 457.45,Z 212.768,A -85,B 0,C 180,E1 -8352.971,E2 -8352.971} C_VEL
LIN {X 0,Y 456.617,Z 300.597,A -85,B 0,C 180,E1 -8354.432,E2 -8354.432} C_VEL
LIN {X 0,Y 456.213,Z 314.412,A -85,B 0,C 180,E1 -8354.847,E2 -8354.847} C_VEL
LIN {X 0,Y 455.753,Z 326.312,A -85,B 0,C 180,E1 -8355.374,E2 -8355.374} C_VEL
LIN {X 0,Y 455.221,Z 337.6,A -85,B 0,C 180,E1 -8356.041,E2 -8356.041} C_VEL
LIN {X 0,Y 454.641,Z 349.738,A -85,B 0,C 180,E1 -8356.973,E2 -8356.973} C_VEL
LIN {X 0,Y 454.137,Z 360.862,A -85,B 0,C 180,E1 -8358.054,E2 -8358.054} C_VEL
LIN {X 0,Y 453.545,Z 370.911,A -85,B 0,C 180,E1 -8359.284,E2 -8359.284} C_VEL
LIN {X 0,Y 453.126,Z 379.763,A -85,B 0,C 180,E1 -8360.627,E2 -8360.627} C_VEL
LIN {X 0,Y 452.842,Z 386.824,A -85,B 0,C 180,E1 -8361.971,E2 -8361.971} C_VEL
LIN {X 0,Y 452.612,Z 393.53,A -85,B 0,C 180,E1 -8363.604,E2 -8363.604} C_VEL
LIN {X 0,Y 452.543,Z 398.146,A -85,B 0,C 180,E1 -8365.1,E2 -8365.1} C_VEL
LIN {X 0,Y 452.48,Z 401.134,A -85,B 0,C 180,E1 -8366.438,E2 -8366.438} C_VEL
LIN {X 0,Y 452.508,Z 402.571,A -85,B 0,C 180,E1 -8367.329,E2 -8367.329} C_VEL
LIN {X 0,Y 452.43,Z 404.205,A -85,B 0,C 180,E1 -8369.11,E2 -8369.11} C_VEL
LIN {X 0,Y 452.437,Z 404.433,A -85,B 0,C 180,E1 -8370,E2 -8370} C_VEL
LIN {X 0,Y 452.43,Z 404.223,A -85,B 0,C 180,E1 -8370.89,E2 -8370.89} C_VEL
LIN {X 0,Y 452.508,Z 402.602,A -85,B 0,C 180,E1 -8372.67,E2 -8372.67} C_VEL
LIN {X 0,Y 452.479,Z 401.189,A -85,B 0,C 180,E1 -8373.562,E2 -8373.562} C_VEL
LIN {X 0,Y 452.543,Z 398.218,A -85,B 0,C 180,E1 -8374.9,E2 -8374.9} C_VEL
LIN {X 0,Y 452.611,Z 393.652,A -85,B 0,C 180,E1 -8376.396,E2 -8376.396} C_VEL
LIN {X 0,Y 452.808,Z 388.011,A -85,B 0,C 180,E1 -8377.805,E2 -8377.805} C_VEL
LIN {X 0,Y 453.08,Z 381.258,A -85,B 0,C 180,E1 -8379.148,E2 -8379.148} C_VEL
LIN {X 0,Y 453.467,Z 372.886,A -85,B 0,C 180,E1 -8380.492,E2 -8380.492} C_VEL
LIN {X 0,Y 453.995,Z 364.291,A -85,B 0,C 180,E1 -8381.609,E2 -8381.609} C_VEL
LIN {X 0,Y 454.611,Z 353.222,A -85,B 0,C 180,E1 -8382.77,E2 -8382.77} C_VEL
LIN {X 0,Y 455.118,Z 341.737,A -85,B 0,C 180,E1 -8383.734,E2 -8383.734} C_VEL
LIN {X 0,Y 455.731,Z 329.682,A -85,B 0,C 180,E1 -8384.512,E2 -8384.512} C_VEL
LIN {X 0,Y 456.274,Z 317.164,A -85,B 0,C 180,E1 -8385.122,E2 -8385.122} C_VEL
LIN {X 0,Y 456.706,Z 305.173,A -85,B 0,C 180,E1 -8385.536,E2 -8385.536} C_VEL
LIN {X 0,Y 456.982,Z 292.159,A -85,B 0,C 180,E1 -8385.813,E2 -8385.813} C_VEL
LIN {X 0,Y 457.611,Z 211.663,A -85,B 0,C 180,E1 -8387.155,E2 -8387.155} C_VEL
LIN {X 0,Y 454.412,Z 191.39,A -85,B 0,C 180,E1 -8387.662,E2 -8387.662} C_VEL
LIN {X 0,Y 455.14,Z 174.094,A -85,B 0,C 180,E1 -8390.802,E2 -8390.802} C_VEL
LIN {X 0,Y 455.855,Z 159.989,A -85,B 0,C 180,E1 -8393.39,E2 -8393.39} C_VEL
LIN {X 0,Y 454.325,Z 150.992,A -85,B 0,C 180,E1 -8395.175,E2 -8395.175} C_VEL
LIN {X 0,Y 453.469,Z 147.001,A -85,B 0,C 180,E1 -8396.017,E2 -8396.017} C_VEL
LIN {X 0,Y 453.447,Z 147.005,A -85,B 0,C 180,E1 -8398.716,E2 -8398.716} C_VEL
LIN {X 0,Y 453.44,Z 147.006,A -85,B 0,C 180,E1 -8401.801,E2 -8401.801} C_VEL
LIN {X 0,Y 453.47,Z 147.002,A -85,B 0,C 180,E1 -8404.989,E2 -8404.989} C_VEL
LIN {X 0,Y 453.442,Z 147.002,A -85,B 0,C 180,E1 -8408.313,E2 -8408.313} C_VEL
LIN {X 0,Y 453.467,Z 147.001,A -85,B 0,C 180,E1 -8410.611,E2 -8410.611} C_VEL
LIN {X 0,Y 453.477,Z 147,A -85,B 0,C 180,E1 -8414.527,E2 -8414.527} C_VEL
LIN {X 0,Y 453.431,Z 146.999,A -85,B 0,C 180,E1 -8418.07,E2 -8418.07} C_VEL
LIN {X 0,Y 453.433,Z 147.003,A -85,B 0,C 180,E1 -8420.802,E2 -8420.802} C_VEL
LIN {X 0,Y 453.437,Z 146.997,A -85,B 0,C 180,E1 -8423.915,E2 -8423.915} C_VEL
LIN {X 0,Y 453.467,Z 146.997,A -85,B 0,C 180,E1 -8427.149,E2 -8427.149} C_VEL
LIN {X 0,Y 453.441,Z 146.999,A -85,B 0,C 180,E1 -8430.265,E2 -8430.265} C_VEL
LIN {X 0,Y 453.434,Z 146.996,A -85,B 0,C 180,E1 -8433.289,E2 -8433.289} C_VEL
LIN {X 0,Y 453.475,Z 147,A -85,B 0,C 180,E1 -8436.237,E2 -8436.237} C_VEL
LIN {X 0,Y 453.452,Z 146.999,A -85,B 0,C 180,E1 -8439.116,E2 -8439.116} C_VEL
LIN {X 0,Y 453.453,Z 146.996,A -85,B 0,C 180,E1 -8441.942,E2 -8441.942} C_VEL
LIN {X 0,Y 453.51,Z 146.99,A -85,B 0,C 180,E1 -8444.725,E2 -8444.725} C_VEL
LIN {X 0,Y 453.537,Z 146.989,A -85,B 0,C 180,E1 -8448.378,E2 -8448.378} C_VEL
LIN {X 0,Y 453.55,Z 146.984,A -85,B 0,C 180,E1 -8451.085,E2 -8451.085} C_VEL
LIN {X 0,Y 453.626,Z 146.98,A -85,B 0,C 180,E1 -8453.774,E2 -8453.774} C_VEL
LIN {X 0,Y 453.694,Z 146.969,A -85,B 0,C 180,E1 -8457.336,E2 -8457.336} C_VEL
LIN {X 0,Y 453.759,Z 146.965,A -85,B 0,C 180,E1 -8460,E2 -8460} C_VEL
LIN {X 0,Y 453.694,Z 146.968,A -85,B 0,C 180,E1 -8462.663,E2 -8462.663} C_VEL
LIN {X 0,Y 453.625,Z 146.98,A -85,B 0,C 180,E1 -8466.226,E2 -8466.226} C_VEL
LIN {X 0,Y 453.549,Z 146.988,A -85,B 0,C 180,E1 -8468.914,E2 -8468.914} C_VEL
LIN {X 0,Y 453.556,Z 146.99,A -85,B 0,C 180,E1 -8472.529,E2 -8472.529} C_VEL
LIN {X 0,Y 453.49,Z 146.999,A -85,B 0,C 180,E1 -8476.089,E2 -8476.089} C_VEL
LIN {X 0,Y 453.509,Z 146.995,A -85,B 0,C 180,E1 -8479.039,E2 -8479.039} C_VEL
LIN {X 0,Y 453.463,Z 147.036,A -85,B 0,C 180,E1 -8481.896,E2 -8481.896} C_VEL
LIN {X 0,Y 455.05,Z 155.305,A -85,B 0,C 180,E1 -8483.675,E2 -8483.675} C_VEL
LIN {X 0,Y 454.718,Z 168.881,A -85,B 0,C 180,E1 -8486.407,E2 -8486.407} C_VEL
LIN {X 0,Y 457.936,Z 185.728,A -85,B 0,C 180,E1 -8486.858,E2 -8486.858} C_VEL
LIN {X 0,Y 456.881,Z 277.15,A -85,B 0,C 180,E1 -8488.402,E2 -8488.402} C_VEL
LIN {X 0,Y 456.535,Z 290.877,A -85,B 0,C 180,E1 -8488.827,E2 -8488.827} C_VEL
LIN {X 0,Y 456.173,Z 302.705,A -85,B 0,C 180,E1 -8489.366,E2 -8489.366} C_VEL
LIN {X 0,Y 455.682,Z 314.469,A -85,B 0,C 180,E1 -8490.085,E2 -8490.085} C_VEL
LIN {X 0,Y 455.051,Z 326.452,A -85,B 0,C 180,E1 -8491.028,E2 -8491.028} C_VEL
LIN {X 0,Y 454.529,Z 336.086,A -85,B 0,C 180,E1 -8491.976,E2 -8491.976} C_VEL
LIN {X 0,Y 454.112,Z 344.875,A -85,B 0,C 180,E1 -8493.035,E2 -8493.035} C_VEL
LIN {X 0,Y 453.563,Z 353.639,A -85,B 0,C 180,E1 -8494.332,E2 -8494.332} C_VEL
LIN {X 0,Y 453.167,Z 361.746,A -85,B 0,C 180,E1 -8495.834,E2 -8495.834} C_VEL
LIN {X 0,Y 452.87,Z 367.677,A -85,B 0,C 180,E1 -8497.245,E2 -8497.245} C_VEL
LIN {X 0,Y 452.698,Z 371.524,A -85,B 0,C 180,E1 -8498.388,E2 -8498.388} C_VEL
LIN {X 0,Y 452.585,Z 374.566,A -85,B 0,C 180,E1 -8499.544,E2 -8499.544} C_VEL
LIN {X 0,Y 452.471,Z 376.911,A -85,B 0,C 180,E1 -8500.72,E2 -8500.72} C_VEL
LIN {X 0,Y 452.365,Z 378.562,A -85,B 0,C 180,E1 -8501.916,E2 -8501.916} C_VEL
LIN {X 0,Y 452.322,Z 379.446,A -85,B 0,C 180,E1 -8503.129,E2 -8503.129} C_VEL
LIN {X 0,Y 452.373,Z 379.581,A -85,B 0,C 180,E1 -8504.387,E2 -8504.387} C_VEL
LIN {X 0,Y 452.377,Z 378.932,A -85,B 0,C 180,E1 -8505.646,E2 -8505.646} C_VEL
LIN {X 0,Y 452.43,Z 377.502,A -85,B 0,C 180,E1 -8506.894,E2 -8506.894} C_VEL
LIN {X 0,Y 452.5,Z 375.104,A -85,B 0,C 180,E1 -8508.202,E2 -8508.202} C_VEL
LIN {X 0,Y 452.664,Z 371.685,A -85,B 0,C 180,E1 -8509.531,E2 -8509.531} C_VEL
LIN {X 0,Y 452.841,Z 367.073,A -85,B 0,C 180,E1 -8510.894,E2 -8510.894} C_VEL
LIN {X 0,Y 453.12,Z 361.058,A -85,B 0,C 180,E1 -8512.28,E2 -8512.28} C_VEL
LIN {X 0,Y 453.477,Z 353.308,A -85,B 0,C 180,E1 -8513.696,E2 -8513.696} C_VEL
LIN {X 0,Y 453.925,Z 345.044,A -85,B 0,C 180,E1 -8514.915,E2 -8514.915} C_VEL
LIN {X 0,Y 454.444,Z 335.716,A -85,B 0,C 180,E1 -8516.037,E2 -8516.037} C_VEL
LIN {X 0,Y 454.959,Z 325.458,A -85,B 0,C 180,E1 -8517.033,E2 -8517.033} C_VEL
LIN {X 0,Y 455.48,Z 314.077,A -85,B 0,C 180,E1 -8517.919,E2 -8517.919} C_VEL
LIN {X 0,Y 455.994,Z 301.831,A -85,B 0,C 180,E1 -8518.657,E2 -8518.657} C_VEL
LIN {X 0,Y 456.37,Z 288.295,A -85,B 0,C 180,E1 -8519.249,E2 -8519.249} C_VEL
LIN {X 0,Y 456.55,Z 281.545,A -85,B 0,C 180,E1 -8519.467,E2 -8519.467} C_VEL
LIN {X 0,Y 455.917,Z 275.834,A -85,B 0,C 180,E1 -8519.646,E2 -8519.646} C_VEL
LIN {X 0,Y 450.57,Z 257.162,A -85,B 0,C 180,E1 -8520.154,E2 -8520.154} C_VEL
LIN {X 0,Y 450.06,Z 251.347,A -85,B 0,C 180,E1 -8520.263,E2 -8520.263} C_VEL
LIN {X 0,Y 450.725,Z 185.449,A -85,B 0,C 180,E1 -8521.367,E2 -8521.367} C_VEL
LIN {X 0,Y 447.574,Z 168.899,A -85,B 0,C 180,E1 -8521.783,E2 -8521.783} C_VEL
LIN {X 0,Y 448.062,Z 157.589,A -85,B 0,C 180,E1 -8524.198,E2 -8524.198} C_VEL
LIN {X 0,Y 446.715,Z 149.202,A -85,B 0,C 180,E1 -8526.102,E2 -8526.102} C_VEL
LIN {X 0,Y 446.447,Z 147.876,A -85,B 0,C 180,E1 -8526.456,E2 -8526.456} C_VEL
LIN {X 0,Y 446.431,Z 147.874,A -85,B 0,C 180,E1 -8529.737,E2 -8529.737} C_VEL
LIN {X 0,Y 446.43,Z 147.878,A -85,B 0,C 180,E1 -8532.596,E2 -8532.596} C_VEL
LIN {X 0,Y 446.451,Z 147.869,A -85,B 0,C 180,E1 -8535.412,E2 -8535.412} C_VEL
LIN {X 0,Y 446.502,Z 147.868,A -85,B 0,C 180,E1 -8538.193,E2 -8538.193} C_VEL
LIN {X 0,Y 446.505,Z 147.863,A -85,B 0,C 180,E1 -8540.944,E2 -8540.944} C_VEL
LIN {X 0,Y 446.6,Z 147.852,A -85,B 0,C 180,E1 -8543.676,E2 -8543.676} C_VEL
LIN {X 0,Y 446.648,Z 147.844,A -85,B 0,C 180,E1 -8547.295,E2 -8547.295} C_VEL
LIN {X 0,Y 446.714,Z 147.843,A -85,B 0,C 180,E1 -8550,E2 -8550} C_VEL
LIN {X 0,Y 446.647,Z 147.845,A -85,B 0,C 180,E1 -8552.706,E2 -8552.706} C_VEL
LIN {X 0,Y 446.6,Z 147.853,A -85,B 0,C 180,E1 -8556.324,E2 -8556.324} C_VEL
LIN {X 0,Y 446.505,Z 147.862,A -85,B 0,C 180,E1 -8559.056,E2 -8559.056} C_VEL
LIN {X 0,Y 446.518,Z 147.86,A -85,B 0,C 180,E1 -8562.73,E2 -8562.73} C_VEL
LIN {X 0,Y 446.446,Z 147.872,A -85,B 0,C 180,E1 -8566.207,E2 -8566.207} C_VEL
LIN {X 0,Y 446.427,Z 147.875,A -85,B 0,C 180,E1 -8569.305,E2 -8569.305} C_VEL
LIN {X 0,Y 446.403,Z 147.876,A -85,B 0,C 180,E1 -8572.2,E2 -8572.2} C_VEL
LIN {X 0,Y 446.416,Z 147.876,A -85,B 0,C 180,E1 -8575.155,E2 -8575.155} C_VEL
LIN {X 0,Y 446.411,Z 147.874,A -85,B 0,C 180,E1 -8578.183,E2 -8578.183} C_VEL
LIN {X 0,Y 446.387,Z 147.883,A -85,B 0,C 180,E1 -8581.302,E2 -8581.302} C_VEL
LIN {X 0,Y 446.416,Z 147.873,A -85,B 0,C 180,E1 -8584.524,E2 -8584.524} C_VEL
LIN {X 0,Y 446.399,Z 147.875,A -85,B 0,C 180,E1 -8588.077,E2 -8588.077} C_VEL
LIN {X 0,Y 446.394,Z 147.881,A -85,B 0,C 180,E1 -8591.394,E2 -8591.394} C_VEL
LIN {X 0,Y 446.444,Z 147.877,A -85,B 0,C 180,E1 -8595.104,E2 -8595.104} C_VEL
LIN {X 0,Y 446.394,Z 147.879,A -85,B 0,C 180,E1 -8598.606,E2 -8598.606} C_VEL
LIN {X 0,Y 446.391,Z 147.876,A -85,B 0,C 180,E1 -8601.924,E2 -8601.924} C_VEL
LIN {X 0,Y 446.413,Z 147.875,A -85,B 0,C 180,E1 -8605.476,E2 -8605.476} C_VEL
LIN {X 0,Y 446.401,Z 147.882,A -85,B 0,C 180,E1 -8608.699,E2 -8608.699} C_VEL
LIN {X 0,Y 446.417,Z 147.873,A -85,B 0,C 180,E1 -8611.836,E2 -8611.836} C_VEL
LIN {X 0,Y 446.414,Z 147.878,A -85,B 0,C 180,E1 -8614.846,E2 -8614.846} C_VEL
LIN {X 0,Y 446.439,Z 147.874,A -85,B 0,C 180,E1 -8618.246,E2 -8618.246} C_VEL
LIN {X 0,Y 446.432,Z 147.871,A -85,B 0,C 180,E1 -8621.649,E2 -8621.649} C_VEL
LIN {X 0,Y 446.452,Z 147.876,A -85,B 0,C 180,E1 -8624.478,E2 -8624.478} C_VEL
LIN {X 0,Y 446.51,Z 147.861,A -85,B 0,C 180,E1 -8627.385,E2 -8627.385} C_VEL
LIN {X 0,Y 446.5,Z 147.864,A -85,B 0,C 180,E1 -8630.944,E2 -8630.944} C_VEL
LIN {X 0,Y 446.597,Z 147.852,A -85,B 0,C 180,E1 -8633.676,E2 -8633.676} C_VEL
LIN {X 0,Y 446.645,Z 147.845,A -85,B 0,C 180,E1 -8637.295,E2 -8637.295} C_VEL
LIN {X 0,Y 446.711,Z 147.843,A -85,B 0,C 180,E1 -8640,E2 -8640} C_VEL
LIN {X 0,Y 446.645,Z 147.845,A -85,B 0,C 180,E1 -8642.706,E2 -8642.706} C_VEL
LIN {X 0,Y 446.598,Z 147.853,A -85,B 0,C 180,E1 -8646.325,E2 -8646.325} C_VEL
LIN {X 0,Y 446.503,Z 147.863,A -85,B 0,C 180,E1 -8649.056,E2 -8649.056} C_VEL
LIN {X 0,Y 446.517,Z 147.861,A -85,B 0,C 180,E1 -8652.73,E2 -8652.73} C_VEL
LIN {X 0,Y 446.445,Z 147.871,A -85,B 0,C 180,E1 -8656.207,E2 -8656.207} C_VEL
LIN {X 0,Y 446.427,Z 147.875,A -85,B 0,C 180,E1 -8659.305,E2 -8659.305} C_VEL
LIN {X 0,Y 446.402,Z 147.876,A -85,B 0,C 180,E1 -8662.201,E2 -8662.201} C_VEL
LIN {X 0,Y 446.416,Z 147.877,A -85,B 0,C 180,E1 -8665.155,E2 -8665.155} C_VEL
LIN {X 0,Y 446.411,Z 147.874,A -85,B 0,C 180,E1 -8668.184,E2 -8668.184} C_VEL
LIN {X 0,Y 446.388,Z 147.884,A -85,B 0,C 180,E1 -8671.303,E2 -8671.303} C_VEL
LIN {X 0,Y 446.416,Z 147.874,A -85,B 0,C 180,E1 -8674.525,E2 -8674.525} C_VEL
LIN {X 0,Y 446.395,Z 147.876,A -85,B 0,C 180,E1 -8678.077,E2 -8678.077} C_VEL
LIN {X 0,Y 446.397,Z 147.88,A -85,B 0,C 180,E1 -8681.395,E2 -8681.395} C_VEL
LIN {X 0,Y 446.447,Z 147.876,A -85,B 0,C 180,E1 -8685.105,E2 -8685.105} C_VEL
LIN {X 0,Y 446.398,Z 147.879,A -85,B 0,C 180,E1 -8688.606,E2 -8688.606} C_VEL
LIN {X 0,Y 446.396,Z 147.876,A -85,B 0,C 180,E1 -8691.925,E2 -8691.925} C_VEL
LIN {X 0,Y 446.419,Z 147.874,A -85,B 0,C 180,E1 -8695.477,E2 -8695.477} C_VEL
LIN {X 0,Y 446.391,Z 147.884,A -85,B 0,C 180,E1 -8698.698,E2 -8698.698} C_VEL
LIN {X 0,Y 446.401,Z 147.877,A -85,B 0,C 180,E1 -8701.842,E2 -8701.842} C_VEL
LIN {X 0,Y 446.436,Z 148.005,A -85,B 0,C 180,E1 -8703.764,E2 -8703.764} C_VEL
LIN {X 0,Y 448.724,Z 159.959,A -85,B 0,C 180,E1 -8706.216,E2 -8706.216} C_VEL
LIN {X 0,Y 448.827,Z 163.772,A -85,B 0,C 180,E1 -8706.955,E2 -8706.955} C_VEL
LIN {X 0,Y 447.901,Z 182.269,A -85,B 0,C 180,E1 -8710.428,E2 -8710.428} C_VEL
LIN {X 0,Y 447.392,Z 192.043,A -85,B 0,C 180,E1 -8712.242,E2 -8712.242} C_VEL
LIN {X 0,Y 450.629,Z 213.487,A -85,B 0,C 180,E1 -8712.735,E2 -8712.735} C_VEL
LIN {X 0,Y 449.724,Z 300.723,A -85,B 0,C 180,E1 -8714.216,E2 -8714.216} C_VEL
LIN {X 0,Y 449.32,Z 314.431,A -85,B 0,C 180,E1 -8714.638,E2 -8714.638} C_VEL
LIN {X 0,Y 448.826,Z 326.823,A -85,B 0,C 180,E1 -8715.201,E2 -8715.201} C_VEL
LIN {X 0,Y 448.212,Z 338.715,A -85,B 0,C 180,E1 -8715.934,E2 -8715.934} C_VEL
LIN {X 0,Y 447.646,Z 350.297,A -85,B 0,C 180,E1 -8716.853,E2 -8716.853} C_VEL
LIN {X 0,Y 447.168,Z 360.5,A -85,B 0,C 180,E1 -8717.865,E2 -8717.865} C_VEL
LIN {X 0,Y 446.538,Z 370.588,A -85,B 0,C 180,E1 -8719.113,E2 -8719.113} C_VEL
LIN {X 0,Y 446.072,Z 379.468,A -85,B 0,C 180,E1 -8720.478,E2 -8720.478} C_VEL
LIN {X 0,Y 445.783,Z 386.559,A -85,B 0,C 180,E1 -8721.843,E2 -8721.843} C_VEL
LIN {X 0,Y 445.554,Z 392.382,A -85,B 0,C 180,E1 -8723.251,E2 -8723.251} C_VEL
LIN {X 0,Y 445.475,Z 396.663,A -85,B 0,C 180,E1 -8724.568,E2 -8724.568} C_VEL
LIN {X 0,Y 445.411,Z 399.006,A -85,B 0,C 180,E1 -8725.475,E2 -8725.475} C_VEL
LIN {X 0,Y 445.378,Z 400.914,A -85,B 0,C 180,E1 -8726.381,E2 -8726.381} C_VEL
LIN {X 0,Y 445.433,Z 402.362,A -85,B 0,C 180,E1 -8727.287,E2 -8727.287} C_VEL
LIN {X 0,Y 445.34,Z 404.004,A -85,B 0,C 180,E1 -8729.096,E2 -8729.096} C_VEL
LIN {X 0,Y 445.345,Z 404.237,A -85,B 0,C 180,E1 -8730,E2 -8730} C_VEL
LIN {X 0,Y 445.34,Z 404.033,A -85,B 0,C 180,E1 -8730.904,E2 -8730.904} C_VEL
LIN {X 0,Y 445.433,Z 402.417,A -85,B 0,C 180,E1 -8732.713,E2 -8732.713} C_VEL
LIN {X 0,Y 445.377,Z 401.007,A -85,B 0,C 180,E1 -8733.619,E2 -8733.619} C_VEL
LIN {X 0,Y 445.471,Z 398.04,A -85,B 0,C 180,E1 -8734.978,E2 -8734.978} C_VEL
LIN {X 0,Y 445.53,Z 393.875,A -85,B 0,C 180,E1 -8736.385,E2 -8736.385} C_VEL
LIN {X 0,Y 445.734,Z 387.85,A -85,B 0,C 180,E1 -8737.93,E2 -8737.93} C_VEL
LIN {X 0,Y 446.054,Z 381.102,A -85,B 0,C 180,E1 -8739.294,E2 -8739.294} C_VEL
LIN {X 0,Y 446.458,Z 372.733,A -85,B 0,C 180,E1 -8740.659,E2 -8740.659} C_VEL
LIN {X 0,Y 447.015,Z 364.153,A -85,B 0,C 180,E1 -8741.793,E2 -8741.793} C_VEL
LIN {X 0,Y 447.624,Z 353.922,A -85,B 0,C 180,E1 -8742.893,E2 -8742.893} C_VEL
LIN {X 0,Y 448.12,Z 343.096,A -85,B 0,C 180,E1 -8743.837,E2 -8743.837} C_VEL
LIN {X 0,Y 448.792,Z 331.616,A -85,B 0,C 180,E1 -8744.626,E2 -8744.626} C_VEL
LIN {X 0,Y 449.287,Z 319.777,A -85,B 0,C 180,E1 -8745.247,E2 -8745.247} C_VEL
LIN {X 0,Y 449.784,Z 307.117,A -85,B 0,C 180,E1 -8745.723,E2 -8745.723} C_VEL
LIN {X 0,Y 450.11,Z 294.26,A -85,B 0,C 180,E1 -8746.031,E2 -8746.031} C_VEL
LIN {X 0,Y 450.88,Z 212.494,A -85,B 0,C 180,E1 -8747.42,E2 -8747.42} C_VEL
LIN {X 0,Y 447.482,Z 191.206,A -85,B 0,C 180,E1 -8747.963,E2 -8747.963} C_VEL
LIN {X 0,Y 448.345,Z 172.717,A -85,B 0,C 180,E1 -8751.373,E2 -8751.373} C_VEL
LIN {X 0,Y 448.942,Z 161.19,A -85,B 0,C 180,E1 -8753.527,E2 -8753.527} C_VEL
LIN {X 0,Y 447.086,Z 150.916,A -85,B 0,C 180,E1 -8755.612,E2 -8755.612} C_VEL
LIN {X 0,Y 446.388,Z 147.884,A -85,B 0,C 180,E1 -8756.27,E2 -8756.27} C_VEL
LIN {X 0,Y 446.407,Z 147.888,A -85,B 0,C 180,E1 -8759.212,E2 -8759.212} C_VEL
LIN {X 0,Y 446.406,Z 147.88,A -85,B 0,C 180,E1 -8762.362,E2 -8762.362} C_VEL
LIN {X 0,Y 446.408,Z 147.88,A -85,B 0,C 180,E1 -8765.626,E2 -8765.626} C_VEL
LIN {X 0,Y 446.396,Z 147.884,A -85,B 0,C 180,E1 -8769.031,E2 -8769.031} C_VEL
LIN {X 0,Y 446.378,Z 147.883,A -85,B 0,C 180,E1 -8772.269,E2 -8772.269} C_VEL
LIN {X 0,Y 446.418,Z 147.879,A -85,B 0,C 180,E1 -8775.107,E2 -8775.107} C_VEL
LIN {X 0,Y 446.395,Z 147.88,A -85,B 0,C 180,E1 -8778.605,E2 -8778.605} C_VEL
LIN {X 0,Y 446.393,Z 147.878,A -85,B 0,C 180,E1 -8781.923,E2 -8781.923} C_VEL
LIN {X 0,Y 446.415,Z 147.874,A -85,B 0,C 180,E1 -8785.475,E2 -8785.475} C_VEL
LIN {X 0,Y 446.386,Z 147.882,A -85,B 0,C 180,E1 -8788.697,E2 -8788.697} C_VEL
LIN {X 0,Y 446.395,Z 147.877,A -85,B 0,C 180,E1 -8791.841,E2 -8791.841} C_VEL
LIN {X 0,Y 446.414,Z 147.878,A -85,B 0,C 180,E1 -8794.845,E2 -8794.845} C_VEL
LIN {X 0,Y 446.438,Z 147.872,A -85,B 0,C 180,E1 -8798.246,E2 -8798.246} C_VEL
LIN {X 0,Y 446.405,Z 147.872,A -85,B 0,C 180,E1 -8801.647,E2 -8801.647} C_VEL
LIN {X 0,Y 446.45,Z 147.87,A -85,B 0,C 180,E1 -8804.477,E2 -8804.477} C_VEL
LIN {X 0,Y 446.509,Z 147.863,A -85,B 0,C 180,E1 -8807.384,E2 -8807.384} C_VEL
LIN {X 0,Y 446.501,Z 147.863,A -85,B 0,C 180,E1 -8810.944,E2 -8810.944} C_VEL
LIN {X 0,Y 446.596,Z 147.855,A -85,B 0,C 180,E1 -8813.675,E2 -8813.675} C_VEL
LIN {X 0,Y 446.643,Z 147.847,A -85,B 0,C 180,E1 -8817.294,E2 -8817.294} C_VEL
LIN {X 0,Y 446.709,Z 147.843,A -85,B 0,C 180,E1 -8820,E2 -8820} C_VEL
LIN {X 0,Y 446.643,Z 147.846,A -85,B 0,C 180,E1 -8822.705,E2 -8822.705} C_VEL
LIN {X 0,Y 446.595,Z 147.855,A -85,B 0,C 180,E1 -8826.324,E2 -8826.324} C_VEL
LIN {X 0,Y 446.5,Z 147.867,A -85,B 0,C 180,E1 -8829.056,E2 -8829.056} C_VEL
LIN {X 0,Y 446.513,Z 147.867,A -85,B 0,C 180,E1 -8832.73,E2 -8832.73} C_VEL
LIN {X 0,Y 446.442,Z 147.877,A -85,B 0,C 180,E1 -8836.207,E2 -8836.207} C_VEL
LIN {X 0,Y 446.459,Z 147.875,A -85,B 0,C 180,E1 -8839.303,E2 -8839.303} C_VEL
LIN {X 0,Y 446.442,Z 147.88,A -85,B 0,C 180,E1 -8841.645,E2 -8841.645} C_VEL
LIN {X 0,Y 448.117,Z 156.682,A -85,B 0,C 180,E1 -8843.573,E2 -8843.573} C_VEL
LIN {X 0,Y 447.785,Z 169.141,A -85,B 0,C 180,E1 -8846.113,E2 -8846.113} C_VEL
LIN {X 0,Y 451.238,Z 186.63,A -85,B 0,C 180,E1 -8846.586,E2 -8846.586} C_VEL
LIN {X 0,Y 450.091,Z 276.957,A -85,B 0,C 180,E1 -8848.138,E2 -8848.138} C_VEL
LIN {X 0,Y 449.721,Z 290.59,A -85,B 0,C 180,E1 -8848.561,E2 -8848.561} C_VEL
LIN {X 0,Y 449.326,Z 303.009,A -85,B 0,C 180,E1 -8849.132,E2 -8849.132} C_VEL
LIN {X 0,Y 448.841,Z 314.039,A -85,B 0,C 180,E1 -8849.811,E2 -8849.811} C_VEL
LIN {X 0,Y 448.214,Z 325.733,A -85,B 0,C 180,E1 -8850.733,E2 -8850.733} C_VEL
LIN {X 0,Y 447.645,Z 335.811,A -85,B 0,C 180,E1 -8851.726,E2 -8851.726} C_VEL
LIN {X 0,Y 447.147,Z 344.965,A -85,B 0,C 180,E1 -8852.837,E2 -8852.837} C_VEL
LIN {X 0,Y 446.618,Z 352.754,A -85,B 0,C 180,E1 -8853.986,E2 -8853.986} C_VEL
LIN {X 0,Y 446.226,Z 360.022,A -85,B 0,C 180,E1 -8855.301,E2 -8855.301} C_VEL
LIN {X 0,Y 445.869,Z 366.625,A -85,B 0,C 180,E1 -8856.796,E2 -8856.796} C_VEL
LIN {X 0,Y 445.597,Z 372.412,A -85,B 0,C 180,E1 -8858.534,E2 -8858.534} C_VEL
LIN {X 0,Y 445.5,Z 374.57,A -85,B 0,C 180,E1 -8859.377,E2 -8859.377} C_VEL
LIN {X 0,Y 445.394,Z 377.284,A -85,B 0,C 180,E1 -8860.765,E2 -8860.765} C_VEL
LIN {X 0,Y 445.263,Z 378.972,A -85,B 0,C 180,E1 -8862.112,E2 -8862.112} C_VEL
LIN {X 0,Y 445.271,Z 379.842,A -85,B 0,C 180,E1 -8863.985,E2 -8863.985} C_VEL
LIN {X 0,Y 445.279,Z 379.42,A -85,B 0,C 180,E1 -8865.255,E2 -8865.255} C_VEL
LIN {X 0,Y 445.3,Z 378.182,A -85,B 0,C 180,E1 -8866.552,E2 -8866.552} C_VEL
LIN {X 0,Y 445.395,Z 376.062,A -85,B 0,C 180,E1 -8867.869,E2 -8867.869} C_VEL
LIN {X 0,Y 445.547,Z 372.954,A -85,B 0,C 180,E1 -8869.213,E2 -8869.213} C_VEL
LIN {X 0,Y 445.763,Z 367.564,A -85,B 0,C 180,E1 -8870.903,E2 -8870.903} C_VEL
LIN {X 0,Y 446.075,Z 361.342,A -85,B 0,C 180,E1 -8872.374,E2 -8872.374} C_VEL
LIN {X 0,Y 446.403,Z 354.482,A -85,B 0,C 180,E1 -8873.666,E2 -8873.666} C_VEL
LIN {X 0,Y 446.922,Z 345.425,A -85,B 0,C 180,E1 -8875.041,E2 -8875.041} C_VEL
LIN {X 0,Y 447.465,Z 336.024,A -85,B 0,C 180,E1 -8876.192,E2 -8876.192} C_VEL
LIN {X 0,Y 448.029,Z 325.412,A -85,B 0,C 180,E1 -8877.236,E2 -8877.236} C_VEL
LIN {X 0,Y 448.521,Z 314.854,A -85,B 0,C 180,E1 -8878.074,E2 -8878.074} C_VEL
LIN {X 0,Y 449.087,Z 302.463,A -85,B 0,C 180,E1 -8878.842,E2 -8878.842} C_VEL
LIN {X 0,Y 449.459,Z 289.537,A -85,B 0,C 180,E1 -8879.426,E2 -8879.426} C_VEL
LIN {X 0,Y 449.821,Z 275.885,A -85,B 0,C 180,E1 -8879.838,E2 -8879.838} C_VEL
LIN {X 0,Y 450.06,Z 251.347,A -85,B 0,C 180,E1 -8880.263,E2 -8880.263} C_VEL
LIN {X 0,Y 449.538,Z 245.536,A -85,B 0,C 180,E1 -8880.38,E2 -8880.38} C_VEL
LIN {X 0,Y 444.169,Z 226.844,A -85,B 0,C 180,E1 -8880.892,E2 -8880.892} C_VEL
LIN {X 0,Y 443.598,Z 221.033,A -85,B 0,C 180,E1 -8881.014,E2 -8881.014} C_VEL
LIN {X 0,Y 443.899,Z 186.251,A -85,B 0,C 180,E1 -8881.614,E2 -8881.614} C_VEL
LIN {X 0,Y 440.639,Z 169.03,A -85,B 0,C 180,E1 -8882.062,E2 -8882.062} C_VEL
LIN {X 0,Y 441.043,Z 157.713,A -85,B 0,C 180,E1 -8884.518,E2 -8884.518} C_VEL
LIN {X 0,Y 439.416,Z 148.753,A -85,B 0,C 180,E1 -8886.619,E2 -8886.619} C_VEL
LIN {X 0,Y 439.377,Z 148.753,A -85,B 0,C 180,E1 -8889.397,E2 -8889.397} C_VEL
LIN {X 0,Y 439.384,Z 148.755,A -85,B 0,C 180,E1 -8892.308,E2 -8892.308} C_VEL
LIN {X 0,Y 439.396,Z 148.748,A -85,B 0,C 180,E1 -8895.173,E2 -8895.173} C_VEL
LIN {X 0,Y 439.472,Z 148.741,A -85,B 0,C 180,E1 -8898.001,E2 -8898.001} C_VEL
LIN {X 0,Y 439.476,Z 148.739,A -85,B 0,C 180,E1 -8901.725,E2 -8901.725} C_VEL
LIN {X 0,Y 439.591,Z 148.727,A -85,B 0,C 180,E1 -8904.496,E2 -8904.496} C_VEL
LIN {X 0,Y 439.623,Z 148.727,A -85,B 0,C 180,E1 -8908.168,E2 -8908.168} C_VEL
LIN {X 0,Y 439.665,Z 148.721,A -85,B 0,C 180,E1 -8910,E2 -8910} C_VEL
LIN {X 0,Y 439.599,Z 148.723,A -85,B 0,C 180,E1 -8912.749,E2 -8912.749} C_VEL
LIN {X 0,Y 439.554,Z 148.73,A -85,B 0,C 180,E1 -8916.426,E2 -8916.426} C_VEL
LIN {X 0,Y 439.471,Z 148.739,A -85,B 0,C 180,E1 -8919.202,E2 -8919.202} C_VEL
LIN {X 0,Y 439.461,Z 148.74,A -85,B 0,C 180,E1 -8922.938,E2 -8922.938} C_VEL
LIN {X 0,Y 439.393,Z 148.749,A -85,B 0,C 180,E1 -8926.326,E2 -8926.326} C_VEL
LIN {X 0,Y 439.373,Z 148.758,A -85,B 0,C 180,E1 -8929.627,E2 -8929.627} C_VEL
LIN {X 0,Y 439.348,Z 148.754,A -85,B 0,C 180,E1 -8932.576,E2 -8932.576} C_VEL
LIN {X 0,Y 439.362,Z 148.759,A -85,B 0,C 180,E1 -8935.587,E2 -8935.587} C_VEL
LIN {X 0,Y 439.372,Z 148.751,A -85,B 0,C 180,E1 -8938.676,E2 -8938.676} C_VEL
LIN {X 0,Y 439.348,Z 148.755,A -85,B 0,C 180,E1 -8942.026,E2 -8942.026} C_VEL
LIN {X 0,Y 439.385,Z 148.756,A -85,B 0,C 180,E1 -8945.339,E2 -8945.339} C_VEL
LIN {X 0,Y 439.352,Z 148.754,A -85,B 0,C 180,E1 -8948.598,E2 -8948.598} C_VEL
LIN {X 0,Y 439.343,Z 148.754,A -85,B 0,C 180,E1 -8952.21,E2 -8952.21} C_VEL
LIN {X 0,Y 439.391,Z 148.753,A -85,B 0,C 180,E1 -8955.27,E2 -8955.27} C_VEL
LIN {X 0,Y 439.348,Z 148.761,A -85,B 0,C 180,E1 -8959.016,E2 -8959.016} C_VEL
LIN {X 0,Y 439.35,Z 148.754,A -85,B 0,C 180,E1 -8961.611,E2 -8961.611} C_VEL
LIN {X 0,Y 439.385,Z 148.757,A -85,B 0,C 180,E1 -8964.843,E2 -8964.843} C_VEL
LIN {X 0,Y 439.359,Z 148.753,A -85,B 0,C 180,E1 -8968.139,E2 -8968.139} C_VEL
LIN {X 0,Y 439.38,Z 148.75,A -85,B 0,C 180,E1 -8971.61,E2 -8971.61} C_VEL
LIN {X 0,Y 439.36,Z 148.757,A -85,B 0,C 180,E1 -8974.413,E2 -8974.413} C_VEL
LIN {X 0,Y 439.347,Z 148.754,A -85,B 0,C 180,E1 -8977.424,E2 -8977.424} C_VEL
LIN {X 0,Y 439.434,Z 148.748,A -85,B 0,C 180,E1 -8980.664,E2 -8980.664} C_VEL
LIN {X 0,Y 439.412,Z 148.751,A -85,B 0,C 180,E1 -8984.223,E2 -8984.223} C_VEL
LIN {X 0,Y 439.478,Z 148.737,A -85,B 0,C 180,E1 -8987.286,E2 -8987.286} C_VEL
LIN {X 0,Y 439.466,Z 148.741,A -85,B 0,C 180,E1 -8990.798,E2 -8990.798} C_VEL
LIN {X 0,Y 439.551,Z 148.729,A -85,B 0,C 180,E1 -8993.574,E2 -8993.574} C_VEL
LIN {X 0,Y 439.397,Z 148.748,A -85,B 0,C 180,E1 -8995.413,E2 -8995.413} C_VEL
LIN {X 0,Y 439.62,Z 148.727,A -85,B 0,C 180,E1 -8998.168,E2 -8998.168} C_VEL
LIN {X 0,Y 439.662,Z 148.721,A -85,B 0,C 180,E1 -9000,E2 -9000} C_VEL
LIN {X 0,Y 439.596,Z 148.723,A -85,B 0,C 180,E1 -9002.749,E2 -9002.749} C_VEL
LIN {X 0,Y 439.551,Z 148.73,A -85,B 0,C 180,E1 -9006.427,E2 -9006.427} C_VEL
LIN {X 0,Y 439.469,Z 148.739,A -85,B 0,C 180,E1 -9009.203,E2 -9009.203} C_VEL
LIN {X 0,Y 439.46,Z 148.74,A -85,B 0,C 180,E1 -9012.938,E2 -9012.938} C_VEL
LIN {X 0,Y 439.392,Z 148.749,A -85,B 0,C 180,E1 -9016.326,E2 -9016.326} C_VEL
LIN {X 0,Y 439.372,Z 148.758,A -85,B 0,C 180,E1 -9019.628,E2 -9019.628} C_VEL
LIN {X 0,Y 439.348,Z 148.754,A -85,B 0,C 180,E1 -9022.577,E2 -9022.577} C_VEL
LIN {X 0,Y 439.362,Z 148.758,A -85,B 0,C 180,E1 -9025.588,E2 -9025.588} C_VEL
LIN {X 0,Y 439.373,Z 148.751,A -85,B 0,C 180,E1 -9028.677,E2 -9028.677} C_VEL
LIN {X 0,Y 439.348,Z 148.754,A -85,B 0,C 180,E1 -9032.027,E2 -9032.027} C_VEL
LIN {X 0,Y 439.384,Z 148.756,A -85,B 0,C 180,E1 -9035.339,E2 -9035.339} C_VEL
LIN {X 0,Y 439.352,Z 148.754,A -85,B 0,C 180,E1 -9038.599,E2 -9038.599} C_VEL
LIN {X 0,Y 439.36,Z 148.758,A -85,B 0,C 180,E1 -9041.253,E2 -9041.253} C_VEL
LIN {X 0,Y 439.395,Z 148.751,A -85,B 0,C 180,E1 -9044.731,E2 -9044.731} C_VEL
LIN {X 0,Y 439.345,Z 148.754,A -85,B 0,C 180,E1 -9047.79,E2 -9047.79} C_VEL
LIN {X 0,Y 439.358,Z 148.753,A -85,B 0,C 180,E1 -9050.22,E2 -9050.22} C_VEL
LIN {X 0,Y 439.364,Z 148.752,A -85,B 0,C 180,E1 -9053.712,E2 -9053.712} C_VEL
LIN {X 0,Y 439.358,Z 148.759,A -85,B 0,C 180,E1 -9057.053,E2 -9057.053} C_VEL
LIN {X 0,Y 439.357,Z 148.755,A -85,B 0,C 180,E1 -9060.273,E2 -9060.273} C_VEL
LIN {X 0,Y 439.413,Z 148.874,A -85,B 0,C 180,E1 -9063.547,E2 -9063.547} C_VEL
LIN {X 0,Y 441.744,Z 160.952,A -85,B 0,C 180,E1 -9066.065,E2 -9066.065} C_VEL
LIN {X 0,Y 441.826,Z 165.851,A -85,B 0,C 180,E1 -9067.027,E2 -9067.027} C_VEL
LIN {X 0,Y 440.875,Z 183.758,A -85,B 0,C 180,E1 -9070.442,E2 -9070.442} C_VEL
LIN {X 0,Y 440.433,Z 191.882,A -85,B 0,C 180,E1 -9071.973,E2 -9071.973} C_VEL
LIN {X 0,Y 443.785,Z 213.814,A -85,B 0,C 180,E1 -9072.489,E2 -9072.489} C_VEL
LIN {X 0,Y 442.842,Z 299.69,A -85,B 0,C 180,E1 -9073.964,E2 -9073.964} C_VEL
LIN {X 0,Y 442.486,Z 312.919,A -85,B 0,C 180,E1 -9074.365,E2 -9074.365} C_VEL
LIN {X 0,Y 441.95,Z 326.23,A -85,B 0,C 180,E1 -9074.965,E2 -9074.965} C_VEL
LIN {X 0,Y 441.303,Z 338.228,A -85,B 0,C 180,E1 -9075.709,E2 -9075.709} C_VEL
LIN {X 0,Y 440.696,Z 349.472,A -85,B 0,C 180,E1 -9076.607,E2 -9076.607} C_VEL
LIN {X 0,Y 440.175,Z 360.117,A -85,B 0,C 180,E1 -9077.67,E2 -9077.67} C_VEL
LIN {X 0,Y 439.546,Z 370.249,A -85,B 0,C 180,E1 -9078.938,E2 -9078.938} C_VEL
LIN {X 0,Y 439.044,Z 379.156,A -85,B 0,C 180,E1 -9080.324,E2 -9080.324} C_VEL
LIN {X 0,Y 438.714,Z 386.28,A -85,B 0,C 180,E1 -9081.71,E2 -9081.71} C_VEL
LIN {X 0,Y 438.496,Z 391.96,A -85,B 0,C 180,E1 -9083.096,E2 -9083.096} C_VEL
LIN {X 0,Y 438.373,Z 396.42,A -85,B 0,C 180,E1 -9084.48,E2 -9084.48} C_VEL
LIN {X 0,Y 438.34,Z 398.772,A -85,B 0,C 180,E1 -9085.402,E2 -9085.402} C_VEL
LIN {X 0,Y 438.28,Z 400.688,A -85,B 0,C 180,E1 -9086.322,E2 -9086.322} C_VEL
LIN {X 0,Y 438.341,Z 402.149,A -85,B 0,C 180,E1 -9087.243,E2 -9087.243} C_VEL
LIN {X 0,Y 438.253,Z 403.802,A -85,B 0,C 180,E1 -9089.081,E2 -9089.081} C_VEL
LIN {X 0,Y 438.256,Z 404.04,A -85,B 0,C 180,E1 -9090,E2 -9090} C_VEL
LIN {X 0,Y 438.253,Z 403.845,A -85,B 0,C 180,E1 -9090.919,E2 -9090.919} C_VEL
LIN {X 0,Y 438.341,Z 402.235,A -85,B 0,C 180,E1 -9092.757,E2 -9092.757} C_VEL
LIN {X 0,Y 438.279,Z 400.829,A -85,B 0,C 180,E1 -9093.677,E2 -9093.677} C_VEL
LIN {X 0,Y 438.38,Z 397.867,A -85,B 0,C 180,E1 -9095.058,E2 -9095.058} C_VEL
LIN {X 0,Y 438.449,Z 393.856,A -85,B 0,C 180,E1 -9096.442,E2 -9096.442} C_VEL
LIN {X 0,Y 438.682,Z 387.694,A -85,B 0,C 180,E1 -9098.058,E2 -9098.058} C_VEL
LIN {X 0,Y 439.024,Z 380.957,A -85,B 0,C 180,E1 -9099.444,E2 -9099.444} C_VEL
LIN {X 0,Y 439.458,Z 372.601,A -85,B 0,C 180,E1 -9100.831,E2 -9100.831} C_VEL
LIN {X 0,Y 440.05,Z 364.04,A -85,B 0,C 180,E1 -9101.983,E2 -9101.983} C_VEL
LIN {X 0,Y 440.646,Z 354.242,A -85,B 0,C 180,E1 -9103.06,E2 -9103.06} C_VEL
LIN {X 0,Y 441.207,Z 343.023,A -85,B 0,C 180,E1 -9104.058,E2 -9104.058} C_VEL
LIN {X 0,Y 441.903,Z 331.599,A -85,B 0,C 180,E1 -9104.859,E2 -9104.859} C_VEL
LIN {X 0,Y 442.46,Z 319.862,A -85,B 0,C 180,E1 -9105.488,E2 -9105.488} C_VEL
LIN {X 0,Y 443.029,Z 306.45,A -85,B 0,C 180,E1 -9105.999,E2 -9105.999} C_VEL
LIN {X 0,Y 443.359,Z 293.324,A -85,B 0,C 180,E1 -9106.312,E2 -9106.312} C_VEL
LIN {X 0,Y 444.13,Z 213.177,A -85,B 0,C 180,E1 -9107.7,E2 -9107.7} C_VEL
LIN {X 0,Y 440.511,Z 191.025,A -85,B 0,C 180,E1 -9108.274,E2 -9108.274} C_VEL
LIN {X 0,Y 441.412,Z 173.916,A -85,B 0,C 180,E1 -9111.481,E2 -9111.481} C_VEL
LIN {X 0,Y 442.01,Z 162.413,A -85,B 0,C 180,E1 -9113.67,E2 -9113.67} C_VEL
LIN {X 0,Y 440.115,Z 152.219,A -85,B 0,C 180,E1 -9115.777,E2 -9115.777} C_VEL
LIN {X 0,Y 439.36,Z 148.76,A -85,B 0,C 180,E1 -9116.558,E2 -9116.558} C_VEL
LIN {X 0,Y 439.356,Z 148.765,A -85,B 0,C 180,E1 -9119.727,E2 -9119.727} C_VEL
LIN {X 0,Y 439.357,Z 148.76,A -85,B 0,C 180,E1 -9122.947,E2 -9122.947} C_VEL
LIN {X 0,Y 439.363,Z 148.755,A -85,B 0,C 180,E1 -9126.287,E2 -9126.287} C_VEL
LIN {X 0,Y 439.357,Z 148.758,A -85,B 0,C 180,E1 -9129.779,E2 -9129.779} C_VEL
LIN {X 0,Y 439.33,Z 148.763,A -85,B 0,C 180,E1 -9132.619,E2 -9132.619} C_VEL
LIN {X 0,Y 439.371,Z 148.757,A -85,B 0,C 180,E1 -9135.266,E2 -9135.266} C_VEL
LIN {X 0,Y 439.349,Z 148.76,A -85,B 0,C 180,E1 -9139.015,E2 -9139.015} C_VEL
LIN {X 0,Y 439.351,Z 148.755,A -85,B 0,C 180,E1 -9141.61,E2 -9141.61} C_VEL
LIN {X 0,Y 439.386,Z 148.756,A -85,B 0,C 180,E1 -9144.842,E2 -9144.842} C_VEL
LIN {X 0,Y 439.348,Z 148.755,A -85,B 0,C 180,E1 -9148.137,E2 -9148.137} C_VEL
LIN {X 0,Y 439.379,Z 148.751,A -85,B 0,C 180,E1 -9151.609,E2 -9151.609} C_VEL
LIN {X 0,Y 439.36,Z 148.754,A -85,B 0,C 180,E1 -9154.412,E2 -9154.412} C_VEL
LIN {X 0,Y 439.346,Z 148.75,A -85,B 0,C 180,E1 -9157.423,E2 -9157.423} C_VEL
LIN {X 0,Y 439.379,Z 148.75,A -85,B 0,C 180,E1 -9160.684,E2 -9160.684} C_VEL
LIN {X 0,Y 439.409,Z 148.749,A -85,B 0,C 180,E1 -9164.222,E2 -9164.222} C_VEL
LIN {X 0,Y 439.477,Z 148.738,A -85,B 0,C 180,E1 -9167.285,E2 -9167.285} C_VEL
LIN {X 0,Y 439.467,Z 148.74,A -85,B 0,C 180,E1 -9170.797,E2 -9170.797} C_VEL
LIN {X 0,Y 439.549,Z 148.732,A -85,B 0,C 180,E1 -9173.573,E2 -9173.573} C_VEL
LIN {X 0,Y 439.395,Z 148.746,A -85,B 0,C 180,E1 -9175.413,E2 -9175.413} C_VEL
LIN {X 0,Y 439.617,Z 148.724,A -85,B 0,C 180,E1 -9178.167,E2 -9178.167} C_VEL
LIN {X 0,Y 439.66,Z 148.72,A -85,B 0,C 180,E1 -9180,E2 -9180} C_VEL
LIN {X 0,Y 439.595,Z 148.724,A -85,B 0,C 180,E1 -9182.749,E2 -9182.749} C_VEL
LIN {X 0,Y 439.549,Z 148.732,A -85,B 0,C 180,E1 -9186.426,E2 -9186.426} C_VEL
LIN {X 0,Y 439.466,Z 148.744,A -85,B 0,C 180,E1 -9189.202,E2 -9189.202} C_VEL
LIN {X 0,Y 439.457,Z 148.747,A -85,B 0,C 180,E1 -9192.937,E2 -9192.937} C_VEL
LIN {X 0,Y 439.389,Z 148.755,A -85,B 0,C 180,E1 -9196.326,E2 -9196.326} C_VEL
LIN {X 0,Y 439.392,Z 148.757,A -85,B 0,C 180,E1 -9199.626,E2 -9199.626} C_VEL
LIN {X 0,Y 439.404,Z 148.808,A -85,B 0,C 180,E1 -9201.399,E2 -9201.399} C_VEL
LIN {X 0,Y 441.19,Z 158.099,A -85,B 0,C 180,E1 -9203.468,E2 -9203.468} C_VEL
LIN {X 0,Y 440.877,Z 169.512,A -85,B 0,C 180,E1 -9205.81,E2 -9205.81} C_VEL
LIN {X 0,Y 444.52,Z 187.133,A -85,B 0,C 180,E1 -9206.297,E2 -9206.297} C_VEL
LIN {X 0,Y 443.304,Z 277.376,A -85,B 0,C 180,E1 -9207.877,E2 -9207.877} C_VEL
LIN {X 0,Y 442.927,Z 291.102,A -85,B 0,C 180,E1 -9208.314,E2 -9208.314} C_VEL
LIN {X 0,Y 442.519,Z 303.042,A -85,B 0,C 180,E1 -9208.873,E2 -9208.873} C_VEL
LIN {X 0,Y 441.917,Z 315.571,A -85,B 0,C 180,E1 -9209.669,E2 -9209.669} C_VEL
LIN {X 0,Y 441.229,Z 327.447,A -85,B 0,C 180,E1 -9210.644,E2 -9210.644} C_VEL
LIN {X 0,Y 440.562,Z 338.159,A -85,B 0,C 180,E1 -9211.764,E2 -9211.764} C_VEL
LIN {X 0,Y 439.988,Z 347.884,A -85,B 0,C 180,E1 -9213.03,E2 -9213.03} C_VEL
LIN {X 0,Y 439.46,Z 355.884,A -85,B 0,C 180,E1 -9214.314,E2 -9214.314} C_VEL
LIN {X 0,Y 439.038,Z 363.158,A -85,B 0,C 180,E1 -9215.777,E2 -9215.777} C_VEL
LIN {X 0,Y 438.77,Z 368.444,A -85,B 0,C 180,E1 -9217.109,E2 -9217.109} C_VEL
LIN {X 0,Y 438.491,Z 373.297,A -85,B 0,C 180,E1 -9218.688,E2 -9218.688} C_VEL
LIN {X 0,Y 438.359,Z 376.049,A -85,B 0,C 180,E1 -9219.888,E2 -9219.888} C_VEL
LIN {X 0,Y 438.269,Z 378.102,A -85,B 0,C 180,E1 -9221.107,E2 -9221.107} C_VEL
LIN {X 0,Y 438.145,Z 379.5,A -85,B 0,C 180,E1 -9222.452,E2 -9222.452} C_VEL
LIN {X 0,Y 438.167,Z 380.015,A -85,B 0,C 180,E1 -9223.8,E2 -9223.8} C_VEL
LIN {X 0,Y 438.193,Z 379.692,A -85,B 0,C 180,E1 -9225.115,E2 -9225.115} C_VEL
LIN {X 0,Y 438.224,Z 378.591,A -85,B 0,C 180,E1 -9226.402,E2 -9226.402} C_VEL
LIN {X 0,Y 438.297,Z 376.739,A -85,B 0,C 180,E1 -9227.666,E2 -9227.666} C_VEL
LIN {X 0,Y 438.426,Z 374.086,A -85,B 0,C 180,E1 -9228.912,E2 -9228.912} C_VEL
LIN {X 0,Y 438.585,Z 370.217,A -85,B 0,C 180,E1 -9230.278,E2 -9230.278} C_VEL
LIN {X 0,Y 438.842,Z 365.033,A -85,B 0,C 180,E1 -9231.695,E2 -9231.695} C_VEL
LIN {X 0,Y 439.172,Z 358.293,A -85,B 0,C 180,E1 -9233.143,E2 -9233.143} C_VEL
LIN {X 0,Y 439.655,Z 349.663,A -85,B 0,C 180,E1 -9234.611,E2 -9234.611} C_VEL
LIN {X 0,Y 440.314,Z 340.178,A -85,B 0,C 180,E1 -9235.901,E2 -9235.901} C_VEL
LIN {X 0,Y 440.854,Z 329.684,A -85,B 0,C 180,E1 -9237.043,E2 -9237.043} C_VEL
LIN {X 0,Y 441.386,Z 319.512,A -85,B 0,C 180,E1 -9237.939,E2 -9237.939} C_VEL
LIN {X 0,Y 441.934,Z 307.819,A -85,B 0,C 180,E1 -9238.758,E2 -9238.758} C_VEL
LIN {X 0,Y 442.465,Z 296.054,A -85,B 0,C 180,E1 -9239.38,E2 -9239.38} C_VEL
LIN {X 0,Y 442.783,Z 283.262,A -85,B 0,C 180,E1 -9239.871,E2 -9239.871} C_VEL
LIN {X 0,Y 443.034,Z 270.183,A -85,B 0,C 180,E1 -9240.185,E2 -9240.185} C_VEL
LIN {X 0,Y 443.598,Z 221.033,A -85,B 0,C 180,E1 -9241.014,E2 -9241.014} C_VEL
LIN {X 0,Y 443.027,Z 215.225,A -85,B 0,C 180,E1 -9241.136,E2 -9241.136} C_VEL
LIN {X 0,Y 437.699,Z 196.549,A -85,B 0,C 180,E1 -9241.67,E2 -9241.67} C_VEL
LIN {X 0,Y 437.21,Z 190.743,A -85,B 0,C 180,E1 -9241.793,E2 -9241.793} C_VEL
LIN {X 0,Y 436.842,Z 185.785,A -85,B 0,C 180,E1 -9241.896,E2 -9241.896} C_VEL
LIN {X 0,Y 433.703,Z 169.234,A -85,B 0,C 180,E1 -9242.332,E2 -9242.332} C_VEL
LIN {X 0,Y 434.07,Z 158.962,A -85,B 0,C 180,E1 -9244.593,E2 -9244.593} C_VEL
LIN {X 0,Y 432.345,Z 149.633,A -85,B 0,C 180,E1 -9246.816,E2 -9246.816} C_VEL
LIN {X 0,Y 432.382,Z 149.629,A -85,B 0,C 180,E1 -9250.516,E2 -9250.516} C_VEL
LIN {X 0,Y 432.384,Z 149.623,A -85,B 0,C 180,E1 -9253.96,E2 -9253.96} C_VEL
LIN {X 0,Y 432.45,Z 149.614,A -85,B 0,C 180,E1 -9257.804,E2 -9257.804} C_VEL
LIN {X 0,Y 432.442,Z 149.615,A -85,B 0,C 180,E1 -9261.59,E2 -9261.59} C_VEL
LIN {X 0,Y 432.566,Z 149.604,A -85,B 0,C 180,E1 -9264.406,E2 -9264.406} C_VEL
LIN {X 0,Y 432.592,Z 149.603,A -85,B 0,C 180,E1 -9268.138,E2 -9268.138} C_VEL
LIN {X 0,Y 432.617,Z 149.599,A -85,B 0,C 180,E1 -9270,E2 -9270} C_VEL
LIN {X 0,Y 432.552,Z 149.601,A -85,B 0,C 180,E1 -9272.794,E2 -9272.794} C_VEL
LIN {X 0,Y 432.51,Z 149.607,A -85,B 0,C 180,E1 -9276.531,E2 -9276.531} C_VEL
LIN {X 0,Y 432.417,Z 149.619,A -85,B 0,C 180,E1 -9279.354,E2 -9279.354} C_VEL
LIN {X 0,Y 432.427,Z 149.616,A -85,B 0,C 180,E1 -9282.803,E2 -9282.803} C_VEL
LIN {X 0,Y 432.352,Z 149.626,A -85,B 0,C 180,E1 -9286.453,E2 -9286.453} C_VEL
LIN {X 0,Y 432.309,Z 149.634,A -85,B 0,C 180,E1 -9289.962,E2 -9289.962} C_VEL
LIN {X 0,Y 432.299,Z 149.633,A -85,B 0,C 180,E1 -9292.965,E2 -9292.965} C_VEL
LIN {X 0,Y 432.313,Z 149.632,A -85,B 0,C 180,E1 -9296.035,E2 -9296.035} C_VEL
LIN {X 0,Y 432.31,Z 149.635,A -85,B 0,C 180,E1 -9299.19,E2 -9299.19} C_VEL
LIN {X 0,Y 432.311,Z 149.63,A -85,B 0,C 180,E1 -9302.444,E2 -9302.444} C_VEL
LIN {X 0,Y 432.33,Z 149.63,A -85,B 0,C 180,E1 -9305.818,E2 -9305.818} C_VEL
LIN {X 0,Y 432.295,Z 149.638,A -85,B 0,C 180,E1 -9309.348,E2 -9309.348} C_VEL
LIN {X 0,Y 432.298,Z 149.633,A -85,B 0,C 180,E1 -9311.801,E2 -9311.801} C_VEL
LIN {X 0,Y 432.328,Z 149.629,A -85,B 0,C 180,E1 -9314.347,E2 -9314.347} C_VEL
LIN {X 0,Y 432.297,Z 149.64,A -85,B 0,C 180,E1 -9317.018,E2 -9317.018} C_VEL
LIN {X 0,Y 432.282,Z 149.634,A -85,B 0,C 180,E1 -9319.828,E2 -9319.828} C_VEL
LIN {X 0,Y 432.29,Z 149.639,A -85,B 0,C 180,E1 -9323.021,E2 -9323.021} C_VEL
LIN {X 0,Y 432.326,Z 149.629,A -85,B 0,C 180,E1 -9326.002,E2 -9326.002} C_VEL
LIN {X 0,Y 432.334,Z 149.628,A -85,B 0,C 180,E1 -9329.492,E2 -9329.492} C_VEL
LIN {X 0,Y 432.313,Z 149.63,A -85,B 0,C 180,E1 -9331.872,E2 -9331.872} C_VEL
LIN {X 0,Y 432.316,Z 149.633,A -85,B 0,C 180,E1 -9334.997,E2 -9334.997} C_VEL
LIN {X 0,Y 432.345,Z 149.628,A -85,B 0,C 180,E1 -9338.046,E2 -9338.046} C_VEL
LIN {X 0,Y 432.374,Z 149.624,A -85,B 0,C 180,E1 -9341.03,E2 -9341.03} C_VEL
LIN {X 0,Y 432.382,Z 149.624,A -85,B 0,C 180,E1 -9343.96,E2 -9343.96} C_VEL
LIN {X 0,Y 432.448,Z 149.615,A -85,B 0,C 180,E1 -9347.804,E2 -9347.804} C_VEL
LIN {X 0,Y 432.439,Z 149.615,A -85,B 0,C 180,E1 -9351.59,E2 -9351.59} C_VEL
LIN {X 0,Y 432.544,Z 149.606,A -85,B 0,C 180,E1 -9354.406,E2 -9354.406} C_VEL
LIN {X 0,Y 432.589,Z 149.603,A -85,B 0,C 180,E1 -9358.138,E2 -9358.138} C_VEL
LIN {X 0,Y 432.614,Z 149.599,A -85,B 0,C 180,E1 -9360,E2 -9360} C_VEL
LIN {X 0,Y 432.55,Z 149.601,A -85,B 0,C 180,E1 -9362.794,E2 -9362.794} C_VEL
LIN {X 0,Y 432.508,Z 149.607,A -85,B 0,C 180,E1 -9366.532,E2 -9366.532} C_VEL
LIN {X 0,Y 432.415,Z 149.619,A -85,B 0,C 180,E1 -9369.354,E2 -9369.354} C_VEL
LIN {X 0,Y 432.426,Z 149.616,A -85,B 0,C 180,E1 -9372.803,E2 -9372.803} C_VEL
LIN {X 0,Y 432.351,Z 149.626,A -85,B 0,C 180,E1 -9376.453,E2 -9376.453} C_VEL
LIN {X 0,Y 432.308,Z 149.634,A -85,B 0,C 180,E1 -9379.962,E2 -9379.962} C_VEL
LIN {X 0,Y 432.299,Z 149.633,A -85,B 0,C 180,E1 -9382.966,E2 -9382.966} C_VEL
LIN {X 0,Y 432.313,Z 149.631,A -85,B 0,C 180,E1 -9386.036,E2 -9386.036} C_VEL
LIN {X 0,Y 432.311,Z 149.635,A -85,B 0,C 180,E1 -9389.19,E2 -9389.19} C_VEL
LIN {X 0,Y 432.312,Z 149.63,A -85,B 0,C 180,E1 -9392.444,E2 -9392.444} C_VEL
LIN {X 0,Y 432.33,Z 149.629,A -85,B 0,C 180,E1 -9395.819,E2 -9395.819} C_VEL
LIN {X 0,Y 432.298,Z 149.637,A -85,B 0,C 180,E1 -9399.349,E2 -9399.349} C_VEL
LIN {X 0,Y 432.3,Z 149.632,A -85,B 0,C 180,E1 -9401.801,E2 -9401.801} C_VEL
LIN {X 0,Y 432.332,Z 149.628,A -85,B 0,C 180,E1 -9404.348,E2 -9404.348} C_VEL
LIN {X 0,Y 432.299,Z 149.639,A -85,B 0,C 180,E1 -9407.019,E2 -9407.019} C_VEL
LIN {X 0,Y 432.287,Z 149.633,A -85,B 0,C 180,E1 -9409.829,E2 -9409.829} C_VEL
LIN {X 0,Y 432.295,Z 149.638,A -85,B 0,C 180,E1 -9413.021,E2 -9413.021} C_VEL
LIN {X 0,Y 432.332,Z 149.628,A -85,B 0,C 180,E1 -9416.003,E2 -9416.003} C_VEL
LIN {X 0,Y 432.331,Z 149.629,A -85,B 0,C 180,E1 -9419.494,E2 -9419.494} C_VEL
LIN {X 0,Y 432.314,Z 149.633,A -85,B 0,C 180,E1 -9421.872,E2 -9421.872} C_VEL
LIN {X 0,Y 432.336,Z 149.697,A -85,B 0,C 180,E1 -9423.311,E2 -9423.311} C_VEL
LIN {X 0,Y 434.735,Z 161.92,A -85,B 0,C 180,E1 -9425.909,E2 -9425.909} C_VEL
LIN {X 0,Y 434.957,Z 165.999,A -85,B 0,C 180,E1 -9426.73,E2 -9426.73} C_VEL
LIN {X 0,Y 433.877,Z 184.741,A -85,B 0,C 180,E1 -9430.36,E2 -9430.36} C_VEL
LIN {X 0,Y 433.459,Z 191.708,A -85,B 0,C 180,E1 -9431.695,E2 -9431.695} C_VEL
LIN {X 0,Y 436.971,Z 215.509,A -85,B 0,C 180,E1 -9432.263,E2 -9432.263} C_VEL
LIN {X 0,Y 435.969,Z 299.657,A -85,B 0,C 180,E1 -9433.734,E2 -9433.734} C_VEL
LIN {X 0,Y 435.574,Z 312.82,A -85,B 0,C 180,E1 -9434.14,E2 -9434.14} C_VEL
LIN {X 0,Y 435.074,Z 325.545,A -85,B 0,C 180,E1 -9434.722,E2 -9434.722} C_VEL
LIN {X 0,Y 434.4,Z 337.691,A -85,B 0,C 180,E1 -9435.477,E2 -9435.477} C_VEL
LIN {X 0,Y 433.713,Z 349.948,A -85,B 0,C 180,E1 -9436.473,E2 -9436.473} C_VEL
LIN {X 0,Y 433.148,Z 360.726,A -85,B 0,C 180,E1 -9437.585,E2 -9437.585} C_VEL
LIN {X 0,Y 432.563,Z 369.894,A -85,B 0,C 180,E1 -9438.757,E2 -9438.757} C_VEL
LIN {X 0,Y 432.024,Z 378.833,A -85,B 0,C 180,E1 -9440.165,E2 -9440.165} C_VEL
LIN {X 0,Y 431.667,Z 385.994,A -85,B 0,C 180,E1 -9441.574,E2 -9441.574} C_VEL
LIN {X 0,Y 431.416,Z 391.696,A -85,B 0,C 180,E1 -9442.982,E2 -9442.982} C_VEL
LIN {X 0,Y 431.275,Z 396.175,A -85,B 0,C 180,E1 -9444.389,E2 -9444.389} C_VEL
LIN {X 0,Y 431.269,Z 398.536,A -85,B 0,C 180,E1 -9445.326,E2 -9445.326} C_VEL
LIN {X 0,Y 431.187,Z 400.459,A -85,B 0,C 180,E1 -9446.262,E2 -9446.262} C_VEL
LIN {X 0,Y 431.236,Z 401.933,A -85,B 0,C 180,E1 -9447.197,E2 -9447.197} C_VEL
LIN {X 0,Y 431.203,Z 402.964,A -85,B 0,C 180,E1 -9448.132,E2 -9448.132} C_VEL
LIN {X 0,Y 431.17,Z 403.842,A -85,B 0,C 180,E1 -9450,E2 -9450} C_VEL
LIN {X 0,Y 431.17,Z 403.657,A -85,B 0,C 180,E1 -9450.934,E2 -9450.934} C_VEL
LIN {X 0,Y 431.203,Z 403.053,A -85,B 0,C 180,E1 -9451.868,E2 -9451.868} C_VEL
LIN {X 0,Y 431.236,Z 402.055,A -85,B 0,C 180,E1 -9452.802,E2 -9452.802} C_VEL
LIN {X 0,Y 431.186,Z 400.654,A -85,B 0,C 180,E1 -9453.738,E2 -9453.738} C_VEL
LIN {X 0,Y 431.291,Z 397.7,A -85,B 0,C 180,E1 -9455.142,E2 -9455.142} C_VEL
LIN {X 0,Y 431.378,Z 393.698,A -85,B 0,C 180,E1 -9456.548,E2 -9456.548} C_VEL
LIN {X 0,Y 431.624,Z 387.549,A -85,B 0,C 180,E1 -9458.191,E2 -9458.191} C_VEL
LIN {X 0,Y 431.972,Z 380.819,A -85,B 0,C 180,E1 -9459.599,E2 -9459.599} C_VEL
LIN {X 0,Y 432.47,Z 372.483,A -85,B 0,C 180,E1 -9461.008,E2 -9461.008} C_VEL
LIN {X 0,Y 433.096,Z 363.952,A -85,B 0,C 180,E1 -9462.178,E2 -9462.178} C_VEL
LIN {X 0,Y 433.686,Z 353.432,A -85,B 0,C 180,E1 -9463.35,E2 -9463.35} C_VEL
LIN {X 0,Y 434.431,Z 341.587,A -85,B 0,C 180,E1 -9464.402,E2 -9464.402} C_VEL
LIN {X 0,Y 435.14,Z 329.719,A -85,B 0,C 180,E1 -9465.215,E2 -9465.215} C_VEL
LIN {X 0,Y 435.788,Z 317.438,A -85,B 0,C 180,E1 -9465.852,E2 -9465.852} C_VEL
LIN {X 0,Y 436.259,Z 305.863,A -85,B 0,C 180,E1 -9466.284,E2 -9466.284} C_VEL
LIN {X 0,Y 436.611,Z 292.426,A -85,B 0,C 180,E1 -9466.601,E2 -9466.601} C_VEL
LIN {X 0,Y 437.459,Z 214.315,A -85,B 0,C 180,E1 -9467.977,E2 -9467.977} C_VEL
LIN {X 0,Y 433.941,Z 192.835,A -85,B 0,C 180,E1 -9468.541,E2 -9468.541} C_VEL
LIN {X 0,Y 433.584,Z 190.721,A -85,B 0,C 180,E1 -9468.622,E2 -9468.622} C_VEL
LIN {X 0,Y 434.554,Z 173.87,A -85,B 0,C 180,E1 -9471.837,E2 -9471.837} C_VEL
LIN {X 0,Y 435.09,Z 163.634,A -85,B 0,C 180,E1 -9473.817,E2 -9473.817} C_VEL
LIN {X 0,Y 433.132,Z 153.406,A -85,B 0,C 180,E1 -9475.982,E2 -9475.982} C_VEL
LIN {X 0,Y 432.314,Z 149.637,A -85,B 0,C 180,E1 -9476.827,E2 -9476.827} C_VEL
LIN {X 0,Y 432.314,Z 149.644,A -85,B 0,C 180,E1 -9479.189,E2 -9479.189} C_VEL
LIN {X 0,Y 432.311,Z 149.637,A -85,B 0,C 180,E1 -9482.443,E2 -9482.443} C_VEL
LIN {X 0,Y 432.331,Z 149.632,A -85,B 0,C 180,E1 -9485.818,E2 -9485.818} C_VEL
LIN {X 0,Y 432.297,Z 149.641,A -85,B 0,C 180,E1 -9489.348,E2 -9489.348} C_VEL
LIN {X 0,Y 432.3,Z 149.637,A -85,B 0,C 180,E1 -9491.8,E2 -9491.8} C_VEL
LIN {X 0,Y 432.329,Z 149.634,A -85,B 0,C 180,E1 -9494.347,E2 -9494.347} C_VEL
LIN {X 0,Y 432.297,Z 149.636,A -85,B 0,C 180,E1 -9497.018,E2 -9497.018} C_VEL
LIN {X 0,Y 432.284,Z 149.634,A -85,B 0,C 180,E1 -9499.827,E2 -9499.827} C_VEL
LIN {X 0,Y 432.291,Z 149.634,A -85,B 0,C 180,E1 -9503.02,E2 -9503.02} C_VEL
LIN {X 0,Y 432.327,Z 149.629,A -85,B 0,C 180,E1 -9506.001,E2 -9506.001} C_VEL
LIN {X 0,Y 432.326,Z 149.627,A -85,B 0,C 180,E1 -9509.493,E2 -9509.493} C_VEL
LIN {X 0,Y 432.308,Z 149.632,A -85,B 0,C 180,E1 -9511.871,E2 -9511.871} C_VEL
LIN {X 0,Y 432.317,Z 149.633,A -85,B 0,C 180,E1 -9514.996,E2 -9514.996} C_VEL
LIN {X 0,Y 432.344,Z 149.625,A -85,B 0,C 180,E1 -9518.045,E2 -9518.045} C_VEL
LIN {X 0,Y 432.336,Z 149.625,A -85,B 0,C 180,E1 -9521.027,E2 -9521.027} C_VEL
LIN {X 0,Y 432.378,Z 149.626,A -85,B 0,C 180,E1 -9523.959,E2 -9523.959} C_VEL
LIN {X 0,Y 432.447,Z 149.617,A -85,B 0,C 180,E1 -9527.803,E2 -9527.803} C_VEL
LIN {X 0,Y 432.439,Z 149.616,A -85,B 0,C 180,E1 -9531.589,E2 -9531.589} C_VEL
LIN {X 0,Y 432.542,Z 149.602,A -85,B 0,C 180,E1 -9534.405,E2 -9534.405} C_VEL
LIN {X 0,Y 432.587,Z 149.6,A -85,B 0,C 180,E1 -9538.138,E2 -9538.138} C_VEL
LIN {X 0,Y 432.612,Z 149.598,A -85,B 0,C 180,E1 -9540,E2 -9540} C_VEL
LIN {X 0,Y 432.548,Z 149.602,A -85,B 0,C 180,E1 -9542.794,E2 -9542.794} C_VEL
LIN {X 0,Y 432.505,Z 149.609,A -85,B 0,C 180,E1 -9546.531,E2 -9546.531} C_VEL
LIN {X 0,Y 432.412,Z 149.625,A -85,B 0,C 180,E1 -9549.353,E2 -9549.353} C_VEL
LIN {X 0,Y 432.423,Z 149.623,A -85,B 0,C 180,E1 -9552.802,E2 -9552.802} C_VEL
LIN {X 0,Y 432.348,Z 149.632,A -85,B 0,C 180,E1 -9556.453,E2 -9556.453} C_VEL
LIN {X 0,Y 432.375,Z 149.63,A -85,B 0,C 180,E1 -9559.483,E2 -9559.483} C_VEL
LIN {X 0,Y 432.373,Z 149.744,A -85,B 0,C 180,E1 -9561.139,E2 -9561.139} C_VEL
LIN {X 0,Y 434.263,Z 159.521,A -85,B 0,C 180,E1 -9563.359,E2 -9563.359} C_VEL
LIN {X 0,Y 433.987,Z 169.554,A -85,B 0,C 180,E1 -9565.467,E2 -9565.467} C_VEL
LIN {X 0,Y 437.794,Z 188.001,A -85,B 0,C 180,E1 -9566.005,E2 -9566.005} C_VEL
LIN {X 0,Y 436.549,Z 277.582,A -85,B 0,C 180,E1 -9567.603,E2 -9567.603} C_VEL
LIN {X 0,Y 436.124,Z 291.172,A -85,B 0,C 180,E1 -9568.04,E2 -9568.04} C_VEL
LIN {X 0,Y 435.727,Z 303.15,A -85,B 0,C 180,E1 -9568.609,E2 -9568.609} C_VEL
LIN {X 0,Y 435.104,Z 315.452,A -85,B 0,C 180,E1 -9569.398,E2 -9569.398} C_VEL
LIN {X 0,Y 434.387,Z 327.051,A -85,B 0,C 180,E1 -9570.356,E2 -9570.356} C_VEL
LIN {X 0,Y 433.763,Z 336.826,A -85,B 0,C 180,E1 -9571.365,E2 -9571.365} C_VEL
LIN {X 0,Y 433.216,Z 345.63,A -85,B 0,C 180,E1 -9572.481,E2 -9572.481} C_VEL
LIN {X 0,Y 432.572,Z 354.019,A -85,B 0,C 180,E1 -9573.778,E2 -9573.778} C_VEL
LIN {X 0,Y 432.144,Z 361.103,A -85,B 0,C 180,E1 -9575.13,E2 -9575.13} C_VEL
LIN {X 0,Y 431.721,Z 367.834,A -85,B 0,C 180,E1 -9576.744,E2 -9576.744} C_VEL
LIN {X 0,Y 431.482,Z 372.58,A -85,B 0,C 180,E1 -9578.239,E2 -9578.239} C_VEL
LIN {X 0,Y 431.269,Z 376.644,A -85,B 0,C 180,E1 -9580.013,E2 -9580.013} C_VEL
LIN {X 0,Y 431.143,Z 378.758,A -85,B 0,C 180,E1 -9581.425,E2 -9581.425} C_VEL
LIN {X 0,Y 431.03,Z 380.119,A -85,B 0,C 180,E1 -9583.221,E2 -9583.221} C_VEL
LIN {X 0,Y 431.091,Z 380.139,A -85,B 0,C 180,E1 -9584.508,E2 -9584.508} C_VEL
LIN {X 0,Y 431.109,Z 379.379,A -85,B 0,C 180,E1 -9585.831,E2 -9585.831} C_VEL
LIN {X 0,Y 431.164,Z 377.774,A -85,B 0,C 180,E1 -9587.18,E2 -9587.18} C_VEL
LIN {X 0,Y 431.27,Z 375.234,A -85,B 0,C 180,E1 -9588.557,E2 -9588.557} C_VEL
LIN {X 0,Y 431.467,Z 371.644,A -85,B 0,C 180,E1 -9589.957,E2 -9589.957} C_VEL
LIN {X 0,Y 431.726,Z 366.824,A -85,B 0,C 180,E1 -9591.387,E2 -9591.387} C_VEL
LIN {X 0,Y 432.075,Z 359.825,A -85,B 0,C 180,E1 -9593,E2 -9593} C_VEL
LIN {X 0,Y 432.532,Z 352.546,A -85,B 0,C 180,E1 -9594.333,E2 -9594.333} C_VEL
LIN {X 0,Y 433.086,Z 343.674,A -85,B 0,C 180,E1 -9595.643,E2 -9595.643} C_VEL
LIN {X 0,Y 433.707,Z 333.231,A -85,B 0,C 180,E1 -9596.886,E2 -9596.886} C_VEL
LIN {X 0,Y 434.301,Z 323.076,A -85,B 0,C 180,E1 -9597.86,E2 -9597.86} C_VEL
LIN {X 0,Y 434.857,Z 311.781,A -85,B 0,C 180,E1 -9598.723,E2 -9598.723} C_VEL
LIN {X 0,Y 435.415,Z 299.582,A -85,B 0,C 180,E1 -9599.441,E2 -9599.441} C_VEL
LIN {X 0,Y 435.806,Z 286.419,A -85,B 0,C 180,E1 -9600.006,E2 -9600.006} C_VEL
LIN {X 0,Y 436.129,Z 273.461,A -85,B 0,C 180,E1 -9600.358,E2 -9600.358} C_VEL
LIN {X 0,Y 437.21,Z 190.743,A -85,B 0,C 180,E1 -9601.793,E2 -9601.793} C_VEL
LIN {X 0,Y 436.66,Z 187.595,A -85,B 0,C 180,E1 -9601.871,E2 -9601.871} C_VEL
LIN {X 0,Y 434.452,Z 183.671,A -85,B 0,C 180,E1 -9602.03,E2 -9602.03} C_VEL
LIN {X 0,Y 428.793,Z 176.361,A -85,B 0,C 180,E1 -9602.393,E2 -9602.393} C_VEL
LIN {X 0,Y 427.364,Z 172.67,A -85,B 0,C 180,E1 -9602.52,E2 -9602.52} C_VEL
LIN {X 0,Y 426.751,Z 169.37,A -85,B 0,C 180,E1 -9602.625,E2 -9602.625} C_VEL
LIN {X 0,Y 427.115,Z 160.198,A -85,B 0,C 180,E1 -9604.671,E2 -9604.671} C_VEL
LIN {X 0,Y 425.299,Z 150.51,A -85,B 0,C 180,E1 -9607.021,E2 -9607.021} C_VEL
LIN {X 0,Y 425.355,Z 150.504,A -85,B 0,C 180,E1 -9610.704,E2 -9610.704} C_VEL
LIN {X 0,Y 425.318,Z 150.502,A -85,B 0,C 180,E1 -9613.686,E2 -9613.686} C_VEL
LIN {X 0,Y 425.389,Z 150.493,A -85,B 0,C 180,E1 -9617.097,E2 -9617.097} C_VEL
LIN {X 0,Y 425.377,Z 150.499,A -85,B 0,C 180,E1 -9620.49,E2 -9620.49} C_VEL
LIN {X 0,Y 425.471,Z 150.482,A -85,B 0,C 180,E1 -9623.36,E2 -9623.36} C_VEL
LIN {X 0,Y 425.34,Z 150.499,A -85,B 0,C 180,E1 -9625.261,E2 -9625.261} C_VEL
LIN {X 0,Y 425.561,Z 150.478,A -85,B 0,C 180,E1 -9628.107,E2 -9628.107} C_VEL
LIN {X 0,Y 425.569,Z 150.477,A -85,B 0,C 180,E1 -9630,E2 -9630} C_VEL
LIN {X 0,Y 425.508,Z 150.478,A -85,B 0,C 180,E1 -9632.84,E2 -9632.84} C_VEL
LIN {X 0,Y 425.472,Z 150.483,A -85,B 0,C 180,E1 -9636.64,E2 -9636.64} C_VEL
LIN {X 0,Y 425.377,Z 150.497,A -85,B 0,C 180,E1 -9639.51,E2 -9639.51} C_VEL
LIN {X 0,Y 425.39,Z 150.493,A -85,B 0,C 180,E1 -9642.903,E2 -9642.903} C_VEL
LIN {X 0,Y 425.31,Z 150.503,A -85,B 0,C 180,E1 -9646.583,E2 -9646.583} C_VEL
LIN {X 0,Y 425.292,Z 150.512,A -85,B 0,C 180,E1 -9649.623,E2 -9649.623} C_VEL
LIN {X 0,Y 425.281,Z 150.507,A -85,B 0,C 180,E1 -9652.339,E2 -9652.339} C_VEL
LIN {X 0,Y 425.255,Z 150.516,A -85,B 0,C 180,E1 -9655.448,E2 -9655.448} C_VEL
LIN {X 0,Y 425.291,Z 150.506,A -85,B 0,C 180,E1 -9658.857,E2 -9658.857} C_VEL
LIN {X 0,Y 425.248,Z 150.512,A -85,B 0,C 180,E1 -9661.928,E2 -9661.928} C_VEL
LIN {X 0,Y 425.289,Z 150.512,A -85,B 0,C 180,E1 -9665.336,E2 -9665.336} C_VEL
LIN {X 0,Y 425.272,Z 150.511,A -85,B 0,C 180,E1 -9668.901,E2 -9668.901} C_VEL
LIN {X 0,Y 425.251,Z 150.512,A -85,B 0,C 180,E1 -9672.655,E2 -9672.655} C_VEL
LIN {X 0,Y 425.279,Z 150.511,A -85,B 0,C 180,E1 -9675.283,E2 -9675.283} C_VEL
LIN {X 0,Y 425.242,Z 150.514,A -85,B 0,C 180,E1 -9678.618,E2 -9678.618} C_VEL
LIN {X 0,Y 425.27,Z 150.513,A -85,B 0,C 180,E1 -9681.099,E2 -9681.099} C_VEL
LIN {X 0,Y 425.286,Z 150.51,A -85,B 0,C 180,E1 -9684.663,E2 -9684.663} C_VEL
LIN {X 0,Y 425.254,Z 150.51,A -85,B 0,C 180,E1 -9688.073,E2 -9688.073} C_VEL
LIN {X 0,Y 425.289,Z 150.506,A -85,B 0,C 180,E1 -9691.365,E2 -9691.365} C_VEL
LIN {X 0,Y 425.253,Z 150.516,A -85,B 0,C 180,E1 -9694.552,E2 -9694.552} C_VEL
LIN {X 0,Y 425.284,Z 150.506,A -85,B 0,C 180,E1 -9697.731,E2 -9697.731} C_VEL
LIN {X 0,Y 425.354,Z 150.502,A -85,B 0,C 180,E1 -9700.704,E2 -9700.704} C_VEL
LIN {X 0,Y 425.316,Z 150.502,A -85,B 0,C 180,E1 -9703.686,E2 -9703.686} C_VEL
LIN {X 0,Y 425.387,Z 150.493,A -85,B 0,C 180,E1 -9707.098,E2 -9707.098} C_VEL
LIN {X 0,Y 425.373,Z 150.499,A -85,B 0,C 180,E1 -9710.49,E2 -9710.49} C_VEL
LIN {X 0,Y 425.469,Z 150.483,A -85,B 0,C 180,E1 -9713.361,E2 -9713.361} C_VEL
LIN {X 0,Y 425.336,Z 150.499,A -85,B 0,C 180,E1 -9715.261,E2 -9715.261} C_VEL
LIN {X 0,Y 425.558,Z 150.479,A -85,B 0,C 180,E1 -9718.108,E2 -9718.108} C_VEL
LIN {X 0,Y 425.566,Z 150.477,A -85,B 0,C 180,E1 -9720,E2 -9720} C_VEL
LIN {X 0,Y 425.505,Z 150.478,A -85,B 0,C 180,E1 -9722.841,E2 -9722.841} C_VEL
LIN {X 0,Y 425.469,Z 150.483,A -85,B 0,C 180,E1 -9726.64,E2 -9726.64} C_VEL
LIN {X 0,Y 425.375,Z 150.498,A -85,B 0,C 180,E1 -9729.51,E2 -9729.51} C_VEL
LIN {X 0,Y 425.388,Z 150.493,A -85,B 0,C 180,E1 -9732.903,E2 -9732.903} C_VEL
LIN {X 0,Y 425.309,Z 150.503,A -85,B 0,C 180,E1 -9736.583,E2 -9736.583} C_VEL
LIN {X 0,Y 425.292,Z 150.512,A -85,B 0,C 180,E1 -9739.623,E2 -9739.623} C_VEL
LIN {X 0,Y 425.281,Z 150.506,A -85,B 0,C 180,E1 -9742.34,E2 -9742.34} C_VEL
LIN {X 0,Y 425.256,Z 150.516,A -85,B 0,C 180,E1 -9745.448,E2 -9745.448} C_VEL
LIN {X 0,Y 425.292,Z 150.506,A -85,B 0,C 180,E1 -9748.858,E2 -9748.858} C_VEL
LIN {X 0,Y 425.249,Z 150.511,A -85,B 0,C 180,E1 -9751.929,E2 -9751.929} C_VEL
LIN {X 0,Y 425.289,Z 150.512,A -85,B 0,C 180,E1 -9755.337,E2 -9755.337} C_VEL
LIN {X 0,Y 425.274,Z 150.511,A -85,B 0,C 180,E1 -9758.902,E2 -9758.902} C_VEL
LIN {X 0,Y 425.253,Z 150.512,A -85,B 0,C 180,E1 -9762.656,E2 -9762.656} C_VEL
LIN {X 0,Y 425.283,Z 150.51,A -85,B 0,C 180,E1 -9765.284,E2 -9765.284} C_VEL
LIN {X 0,Y 425.246,Z 150.514,A -85,B 0,C 180,E1 -9768.619,E2 -9768.619} C_VEL
LIN {X 0,Y 425.275,Z 150.512,A -85,B 0,C 180,E1 -9771.099,E2 -9771.099} C_VEL
LIN {X 0,Y 425.292,Z 150.51,A -85,B 0,C 180,E1 -9774.664,E2 -9774.664} C_VEL
LIN {X 0,Y 425.251,Z 150.51,A -85,B 0,C 180,E1 -9778.072,E2 -9778.072} C_VEL
LIN {X 0,Y 425.292,Z 150.508,A -85,B 0,C 180,E1 -9781.365,E2 -9781.365} C_VEL
LIN {X 0,Y 425.289,Z 150.689,A -85,B 0,C 180,E1 -9783.111,E2 -9783.111} C_VEL
LIN {X 0,Y 427.736,Z 162.883,A -85,B 0,C 180,E1 -9785.747,E2 -9785.747} C_VEL
LIN {X 0,Y 428.015,Z 166.713,A -85,B 0,C 180,E1 -9786.536,E2 -9786.536} C_VEL
LIN {X 0,Y 426.891,Z 185.704,A -85,B 0,C 180,E1 -9790.276,E2 -9790.276} C_VEL
LIN {X 0,Y 426.505,Z 191.52,A -85,B 0,C 180,E1 -9791.407,E2 -9791.407} C_VEL
LIN {X 0,Y 430.166,Z 216.238,A -85,B 0,C 180,E1 -9792.011,E2 -9792.011} C_VEL
LIN {X 0,Y 429.114,Z 299.563,A -85,B 0,C 180,E1 -9793.498,E2 -9793.498} C_VEL
LIN {X 0,Y 428.736,Z 311.931,A -85,B 0,C 180,E1 -9793.88,E2 -9793.88} C_VEL
LIN {X 0,Y 428.191,Z 324.833,A -85,B 0,C 180,E1 -9794.47,E2 -9794.47} C_VEL
LIN {X 0,Y 427.521,Z 337.142,A -85,B 0,C 180,E1 -9795.238,E2 -9795.238} C_VEL
LIN {X 0,Y 426.811,Z 348.323,A -85,B 0,C 180,E1 -9796.144,E2 -9796.144} C_VEL
LIN {X 0,Y 426.168,Z 359.274,A -85,B 0,C 180,E1 -9797.258,E2 -9797.258} C_VEL
LIN {X 0,Y 425.672,Z 367.85,A -85,B 0,C 180,E1 -9798.331,E2 -9798.331} C_VEL
LIN {X 0,Y 425.107,Z 375.746,A -85,B 0,C 180,E1 -9799.522,E2 -9799.522} C_VEL
LIN {X 0,Y 424.698,Z 383.451,A -85,B 0,C 180,E1 -9800.955,E2 -9800.955} C_VEL
LIN {X 0,Y 424.409,Z 389.639,A -85,B 0,C 180,E1 -9802.387,E2 -9802.387} C_VEL
LIN {X 0,Y 424.233,Z 394.22,A -85,B 0,C 180,E1 -9803.713,E2 -9803.713} C_VEL
LIN {X 0,Y 424.198,Z 398.293,A -85,B 0,C 180,E1 -9805.248,E2 -9805.248} C_VEL
LIN {X 0,Y 424.098,Z 400.224,A -85,B 0,C 180,E1 -9806.199,E2 -9806.199} C_VEL
LIN {X 0,Y 424.132,Z 401.714,A -85,B 0,C 180,E1 -9807.15,E2 -9807.15} C_VEL
LIN {X 0,Y 424.129,Z 402.752,A -85,B 0,C 180,E1 -9808.101,E2 -9808.101} C_VEL
LIN {X 0,Y 424.087,Z 403.643,A -85,B 0,C 180,E1 -9810,E2 -9810} C_VEL
LIN {X 0,Y 424.089,Z 403.47,A -85,B 0,C 180,E1 -9810.949,E2 -9810.949} C_VEL
LIN {X 0,Y 424.129,Z 402.872,A -85,B 0,C 180,E1 -9811.899,E2 -9811.899} C_VEL
LIN {X 0,Y 424.131,Z 401.877,A -85,B 0,C 180,E1 -9812.849,E2 -9812.849} C_VEL
LIN {X 0,Y 424.097,Z 400.48,A -85,B 0,C 180,E1 -9813.801,E2 -9813.801} C_VEL
LIN {X 0,Y 424.203,Z 397.537,A -85,B 0,C 180,E1 -9815.228,E2 -9815.228} C_VEL
LIN {X 0,Y 424.302,Z 393.549,A -85,B 0,C 180,E1 -9816.658,E2 -9816.658} C_VEL
LIN {X 0,Y 424.58,Z 387.423,A -85,B 0,C 180,E1 -9818.328,E2 -9818.328} C_VEL
LIN {X 0,Y 424.948,Z 380.714,A -85,B 0,C 180,E1 -9819.76,E2 -9819.76} C_VEL
LIN {X 0,Y 425.462,Z 372.391,A -85,B 0,C 180,E1 -9821.191,E2 -9821.191} C_VEL
LIN {X 0,Y 426.151,Z 363.883,A -85,B 0,C 180,E1 -9822.38,E2 -9822.38} C_VEL
LIN {X 0,Y 426.709,Z 354.211,A -85,B 0,C 180,E1 -9823.488,E2 -9823.488} C_VEL
LIN {X 0,Y 427.444,Z 343.013,A -85,B 0,C 180,E1 -9824.521,E2 -9824.521} C_VEL
LIN {X 0,Y 428.189,Z 331.684,A -85,B 0,C 180,E1 -9825.347,E2 -9825.347} C_VEL
LIN {X 0,Y 428.84,Z 320.171,A -85,B 0,C 180,E1 -9825.993,E2 -9825.993} C_VEL
LIN {X 0,Y 429.442,Z 307.069,A -85,B 0,C 180,E1 -9826.52,E2 -9826.52} C_VEL
LIN {X 0,Y 429.804,Z 294.668,A -85,B 0,C 180,E1 -9826.841,E2 -9826.841} C_VEL
LIN {X 0,Y 430.692,Z 214.691,A -85,B 0,C 180,E1 -9828.286,E2 -9828.286} C_VEL
LIN {X 0,Y 427.335,Z 194.174,A -85,B 0,C 180,E1 -9828.841,E2 -9828.841} C_VEL
LIN {X 0,Y 426.705,Z 190.544,A -85,B 0,C 180,E1 -9828.958,E2 -9828.958} C_VEL
LIN {X 0,Y 427.724,Z 173.823,A -85,B 0,C 180,E1 -9832.204,E2 -9832.204} C_VEL
LIN {X 0,Y 428.166,Z 164.883,A -85,B 0,C 180,E1 -9833.969,E2 -9833.969} C_VEL
LIN {X 0,Y 425.868,Z 153.403,A -85,B 0,C 180,E1 -9836.459,E2 -9836.459} C_VEL
LIN {X 0,Y 425.239,Z 150.52,A -85,B 0,C 180,E1 -9837.146,E2 -9837.146} C_VEL
LIN {X 0,Y 425.27,Z 150.52,A -85,B 0,C 180,E1 -9839.72,E2 -9839.72} C_VEL
LIN {X 0,Y 425.264,Z 150.516,A -85,B 0,C 180,E1 -9843.049,E2 -9843.049} C_VEL
LIN {X 0,Y 425.274,Z 150.511,A -85,B 0,C 180,E1 -9845.927,E2 -9845.927} C_VEL
LIN {X 0,Y 425.255,Z 150.517,A -85,B 0,C 180,E1 -9849.036,E2 -9849.036} C_VEL
LIN {X 0,Y 425.253,Z 150.516,A -85,B 0,C 180,E1 -9852.655,E2 -9852.655} C_VEL
LIN {X 0,Y 425.28,Z 150.512,A -85,B 0,C 180,E1 -9855.283,E2 -9855.283} C_VEL
LIN {X 0,Y 425.243,Z 150.515,A -85,B 0,C 180,E1 -9858.617,E2 -9858.617} C_VEL
LIN {X 0,Y 425.272,Z 150.513,A -85,B 0,C 180,E1 -9861.098,E2 -9861.098} C_VEL
LIN {X 0,Y 425.288,Z 150.51,A -85,B 0,C 180,E1 -9864.663,E2 -9864.663} C_VEL
LIN {X 0,Y 425.247,Z 150.511,A -85,B 0,C 180,E1 -9868.071,E2 -9868.071} C_VEL
LIN {X 0,Y 425.286,Z 150.507,A -85,B 0,C 180,E1 -9871.364,E2 -9871.364} C_VEL
LIN {X 0,Y 425.253,Z 150.512,A -85,B 0,C 180,E1 -9874.552,E2 -9874.552} C_VEL
LIN {X 0,Y 425.283,Z 150.502,A -85,B 0,C 180,E1 -9877.73,E2 -9877.73} C_VEL
LIN {X 0,Y 425.317,Z 150.501,A -85,B 0,C 180,E1 -9880.701,E2 -9880.701} C_VEL
LIN {X 0,Y 425.312,Z 150.505,A -85,B 0,C 180,E1 -9883.685,E2 -9883.685} C_VEL
LIN {X 0,Y 425.386,Z 150.494,A -85,B 0,C 180,E1 -9887.097,E2 -9887.097} C_VEL
LIN {X 0,Y 425.373,Z 150.498,A -85,B 0,C 180,E1 -9890.49,E2 -9890.49} C_VEL
LIN {X 0,Y 425.467,Z 150.485,A -85,B 0,C 180,E1 -9893.36,E2 -9893.36} C_VEL
LIN {X 0,Y 425.334,Z 150.497,A -85,B 0,C 180,E1 -9895.261,E2 -9895.261} C_VEL
LIN {X 0,Y 425.556,Z 150.475,A -85,B 0,C 180,E1 -9898.107,E2 -9898.107} C_VEL
LIN {X 0,Y 425.564,Z 150.476,A -85,B 0,C 180,E1 -9900,E2 -9900} C_VEL
LIN {X 0,Y 425.504,Z 150.48,A -85,B 0,C 180,E1 -9902.84,E2 -9902.84} C_VEL
LIN {X 0,Y 425.467,Z 150.486,A -85,B 0,C 180,E1 -9906.639,E2 -9906.639} C_VEL
LIN {X 0,Y 425.373,Z 150.502,A -85,B 0,C 180,E1 -9909.51,E2 -9909.51} C_VEL
LIN {X 0,Y 425.385,Z 150.501,A -85,B 0,C 180,E1 -9912.903,E2 -9912.903} C_VEL
LIN {X 0,Y 425.306,Z 150.509,A -85,B 0,C 180,E1 -9916.583,E2 -9916.583} C_VEL
LIN {X 0,Y 425.317,Z 150.51,A -85,B 0,C 180,E1 -9919.634,E2 -9919.634} C_VEL
LIN {X 0,Y 425.332,Z 150.706,A -85,B 0,C 180,E1 -9920.872,E2 -9920.872} C_VEL
LIN {X 0,Y 427.355,Z 160.967,A -85,B 0,C 180,E1 -9923.246,E2 -9923.246} C_VEL
LIN {X 0,Y 427.133,Z 169.734,A -85,B 0,C 180,E1 -9925.118,E2 -9925.118} C_VEL
LIN {X 0,Y 431.089,Z 188.672,A -85,B 0,C 180,E1 -9925.693,E2 -9925.693} C_VEL
LIN {X 0,Y 429.808,Z 277.863,A -85,B 0,C 180,E1 -9927.322,E2 -9927.322} C_VEL
LIN {X 0,Y 429.37,Z 291.336,A -85,B 0,C 180,E1 -9927.763,E2 -9927.763} C_VEL
LIN {X 0,Y 428.911,Z 303.874,A -85,B 0,C 180,E1 -9928.371,E2 -9928.371} C_VEL
LIN {X 0,Y 428.329,Z 314.872,A -85,B 0,C 180,E1 -9929.083,E2 -9929.083} C_VEL
LIN {X 0,Y 427.549,Z 326.975,A -85,B 0,C 180,E1 -9930.089,E2 -9930.089} C_VEL
LIN {X 0,Y 426.832,Z 337.63,A -85,B 0,C 180,E1 -9931.211,E2 -9931.211} C_VEL
LIN {X 0,Y 426.214,Z 346.739,A -85,B 0,C 180,E1 -9932.405,E2 -9932.405} C_VEL
LIN {X 0,Y 425.598,Z 354.198,A -85,B 0,C 180,E1 -9933.586,E2 -9933.586} C_VEL
LIN {X 0,Y 425.105,Z 361.833,A -85,B 0,C 180,E1 -9935.075,E2 -9935.075} C_VEL
LIN {X 0,Y 424.707,Z 367.895,A -85,B 0,C 180,E1 -9936.564,E2 -9936.564} C_VEL
LIN {X 0,Y 424.514,Z 371.791,A -85,B 0,C 180,E1 -9937.774,E2 -9937.774} C_VEL
LIN {X 0,Y 424.309,Z 374.967,A -85,B 0,C 180,E1 -9939.006,E2 -9939.006} C_VEL
LIN {X 0,Y 424.166,Z 377.565,A -85,B 0,C 180,E1 -9940.345,E2 -9940.345} C_VEL
LIN {X 0,Y 424.012,Z 379.399,A -85,B 0,C 180,E1 -9941.767,E2 -9941.767} C_VEL
LIN {X 0,Y 423.933,Z 380.307,A -85,B 0,C 180,E1 -9943.162,E2 -9943.162} C_VEL
LIN {X 0,Y 423.993,Z 380.326,A -85,B 0,C 180,E1 -9944.541,E2 -9944.541} C_VEL
LIN {X 0,Y 424.011,Z 379.537,A -85,B 0,C 180,E1 -9945.882,E2 -9945.882} C_VEL
LIN {X 0,Y 424.069,Z 377.989,A -85,B 0,C 180,E1 -9947.198,E2 -9947.198} C_VEL
LIN {X 0,Y 424.183,Z 375.691,A -85,B 0,C 180,E1 -9948.492,E2 -9948.492} C_VEL
LIN {X 0,Y 424.359,Z 372.583,A -85,B 0,C 180,E1 -9949.768,E2 -9949.768} C_VEL
LIN {X 0,Y 424.636,Z 367.44,A -85,B 0,C 180,E1 -9951.375,E2 -9951.375} C_VEL
LIN {X 0,Y 424.999,Z 360.522,A -85,B 0,C 180,E1 -9953.017,E2 -9953.017} C_VEL
LIN {X 0,Y 425.456,Z 353.319,A -85,B 0,C 180,E1 -9954.377,E2 -9954.377} C_VEL
LIN {X 0,Y 426.078,Z 344.397,A -85,B 0,C 180,E1 -9955.737,E2 -9955.737} C_VEL
LIN {X 0,Y 426.698,Z 334.634,A -85,B 0,C 180,E1 -9956.936,E2 -9956.936} C_VEL
LIN {X 0,Y 427.285,Z 324.315,A -85,B 0,C 180,E1 -9957.965,E2 -9957.965} C_VEL
LIN {X 0,Y 427.921,Z 312.458,A -85,B 0,C 180,E1 -9958.902,E2 -9958.902} C_VEL
LIN {X 0,Y 428.54,Z 299.787,A -85,B 0,C 180,E1 -9959.663,E2 -9959.663} C_VEL
LIN {X 0,Y 428.936,Z 286.602,A -85,B 0,C 180,E1 -9960.239,E2 -9960.239} C_VEL
LIN {X 0,Y 429.294,Z 273.335,A -85,B 0,C 180,E1 -9960.602,E2 -9960.602} C_VEL
LIN {X 0,Y 430.336,Z 188.385,A -85,B 0,C 180,E1 -9962.11,E2 -9962.11} C_VEL
LIN {X 0,Y 427.364,Z 172.67,A -85,B 0,C 180,E1 -9962.52,E2 -9962.52} C_VEL
LIN {X 0,Y 426.743,Z 170.482,A -85,B 0,C 180,E1 -9962.65,E2 -9962.65} C_VEL
LIN {X 0,Y 425.311,Z 167.802,A -85,B 0,C 180,E1 -9963.044,E2 -9963.044} C_VEL
LIN {X 0,Y 421.59,Z 162.722,A -85,B 0,C 180,E1 -9964.426,E2 -9964.426} C_VEL
LIN {X 0,Y 419.701,Z 158.422,A -85,B 0,C 180,E1 -9965.484,E2 -9965.484} C_VEL
LIN {X 0,Y 419.152,Z 156.176,A -85,B 0,C 180,E1 -9966.018,E2 -9966.018} C_VEL
LIN {X 0,Y 418.248,Z 151.388,A -85,B 0,C 180,E1 -9967.2,E2 -9967.2} C_VEL
LIN {X 0,Y 418.278,Z 151.384,A -85,B 0,C 180,E1 -9970.364,E2 -9970.364} C_VEL
LIN {X 0,Y 418.275,Z 151.379,A -85,B 0,C 180,E1 -9973.403,E2 -9973.403} C_VEL
LIN {X 0,Y 418.342,Z 151.372,A -85,B 0,C 180,E1 -9977,E2 -9977} C_VEL
LIN {X 0,Y 418.318,Z 151.381,A -85,B 0,C 180,E1 -9980.328,E2 -9980.328} C_VEL
LIN {X 0,Y 418.437,Z 151.359,A -85,B 0,C 180,E1 -9983.248,E2 -9983.248} C_VEL
LIN {X 0,Y 418.312,Z 151.374,A -85,B 0,C 180,E1 -9985.181,E2 -9985.181} C_VEL
LIN {X 0,Y 418.53,Z 151.354,A -85,B 0,C 180,E1 -9988.076,E2 -9988.076} C_VEL
LIN {X 0,Y 418.403,Z 151.363,A -85,B 0,C 180,E1 -9990.963,E2 -9990.963} C_VEL
LIN {X 0,Y 418.465,Z 151.355,A -85,B 0,C 180,E1 -9992.888,E2 -9992.888} C_VEL
LIN {X 0,Y 418.465,Z 151.36,A -85,B 0,C 180,E1 -9995.783,E2 -9995.783} C_VEL
LIN {X 0,Y 418.363,Z 151.368,A -85,B 0,C 180,E1 -9998.696,E2 -9998.696} C_VEL
LIN {X 0,Y 418.35,Z 151.37,A -85,B 0,C 180,E1 -10002.615,E2 -10002.615} C_VEL
LIN {X 0,Y 418.245,Z 151.388,A -85,B 0,C 180,E1 -10005.596,E2 -10005.596} C_VEL
LIN {X 0,Y 418.233,Z 151.384,A -85,B 0,C 180,E1 -10008.619,E2 -10008.619} C_VEL
LIN {X 0,Y 418.222,Z 151.392,A -85,B 0,C 180,E1 -10011.697,E2 -10011.697} C_VEL
LIN {X 0,Y 418.24,Z 151.384,A -85,B 0,C 180,E1 -10014.852,E2 -10014.852} C_VEL
LIN {X 0,Y 418.198,Z 151.39,A -85,B 0,C 180,E1 -10018.07,E2 -10018.07} C_VEL
LIN {X 0,Y 418.23,Z 151.387,A -85,B 0,C 180,E1 -10021.018,E2 -10021.018} C_VEL
LIN {X 0,Y 418.227,Z 151.388,A -85,B 0,C 180,E1 -10023.679,E2 -10023.679} C_VEL
LIN {X 0,Y 418.231,Z 151.391,A -85,B 0,C 180,E1 -10027.225,E2 -10027.225} C_VEL
LIN {X 0,Y 418.201,Z 151.392,A -85,B 0,C 180,E1 -10030.867,E2 -10030.867} C_VEL
LIN {X 0,Y 418.197,Z 151.39,A -85,B 0,C 180,E1 -10033.728,E2 -10033.728} C_VEL
LIN {X 0,Y 418.194,Z 151.39,A -85,B 0,C 180,E1 -10036.447,E2 -10036.447} C_VEL
LIN {X 0,Y 418.201,Z 151.393,A -85,B 0,C 180,E1 -10039.133,E2 -10039.133} C_VEL
LIN {X 0,Y 418.227,Z 151.391,A -85,B 0,C 180,E1 -10042.775,E2 -10042.775} C_VEL
LIN {X 0,Y 418.226,Z 151.387,A -85,B 0,C 180,E1 -10046.321,E2 -10046.321} C_VEL
LIN {X 0,Y 418.232,Z 151.384,A -85,B 0,C 180,E1 -10049.727,E2 -10049.727} C_VEL
LIN {X 0,Y 418.204,Z 151.391,A -85,B 0,C 180,E1 -10053.017,E2 -10053.017} C_VEL
LIN {X 0,Y 418.248,Z 151.385,A -85,B 0,C 180,E1 -10056.217,E2 -10056.217} C_VEL
LIN {X 0,Y 418.239,Z 151.383,A -85,B 0,C 180,E1 -10059.337,E2 -10059.337} C_VEL
LIN {X 0,Y 418.249,Z 151.389,A -85,B 0,C 180,E1 -10062.395,E2 -10062.395} C_VEL
LIN {X 0,Y 418.271,Z 151.379,A -85,B 0,C 180,E1 -10065.402,E2 -10065.402} C_VEL
LIN {X 0,Y 418.296,Z 151.383,A -85,B 0,C 180,E1 -10068.369,E2 -10068.369} C_VEL
LIN {X 0,Y 418.441,Z 151.365,A -85,B 0,C 180,E1 -10072.278,E2 -10072.278} C_VEL
LIN {X 0,Y 418.462,Z 151.363,A -85,B 0,C 180,E1 -10074.217,E2 -10074.217} C_VEL
LIN {X 0,Y 418.527,Z 151.355,A -85,B 0,C 180,E1 -10078.076,E2 -10078.076} C_VEL
LIN {X 0,Y 418.4,Z 151.363,A -85,B 0,C 180,E1 -10080.963,E2 -10080.963} C_VEL
LIN {X 0,Y 418.462,Z 151.356,A -85,B 0,C 180,E1 -10082.888,E2 -10082.888} C_VEL
LIN {X 0,Y 418.435,Z 151.359,A -85,B 0,C 180,E1 -10086.752,E2 -10086.752} C_VEL
LIN {X 0,Y 418.316,Z 151.379,A -85,B 0,C 180,E1 -10089.672,E2 -10089.672} C_VEL
LIN {X 0,Y 418.341,Z 151.371,A -85,B 0,C 180,E1 -10093,E2 -10093} C_VEL
LIN {X 0,Y 418.252,Z 151.382,A -85,B 0,C 180,E1 -10096.71,E2 -10096.71} C_VEL
LIN {X 0,Y 418.237,Z 151.389,A -85,B 0,C 180,E1 -10099.779,E2 -10099.779} C_VEL
LIN {X 0,Y 418.221,Z 151.386,A -85,B 0,C 180,E1 -10102.738,E2 -10102.738} C_VEL
LIN {X 0,Y 418.214,Z 151.389,A -85,B 0,C 180,E1 -10105.908,E2 -10105.908} C_VEL
LIN {X 0,Y 418.251,Z 151.386,A -85,B 0,C 180,E1 -10109.163,E2 -10109.163} C_VEL
LIN {X 0,Y 418.245,Z 151.385,A -85,B 0,C 180,E1 -10112.842,E2 -10112.842} C_VEL
LIN {X 0,Y 418.236,Z 151.384,A -85,B 0,C 180,E1 -10116.237,E2 -10116.237} C_VEL
LIN {X 0,Y 418.196,Z 151.39,A -85,B 0,C 180,E1 -10119.689,E2 -10119.689} C_VEL
LIN {X 0,Y 418.205,Z 151.388,A -85,B 0,C 180,E1 -10122.318,E2 -10122.318} C_VEL
LIN {X 0,Y 418.235,Z 151.39,A -85,B 0,C 180,E1 -10125.109,E2 -10125.109} C_VEL
LIN {X 0,Y 418.217,Z 151.386,A -85,B 0,C 180,E1 -10127.764,E2 -10127.764} C_VEL
LIN {X 0,Y 418.233,Z 151.385,A -85,B 0,C 180,E1 -10131.557,E2 -10131.557} C_VEL
LIN {X 0,Y 418.249,Z 151.385,A -85,B 0,C 180,E1 -10135.158,E2 -10135.158} C_VEL
LIN {X 0,Y 418.237,Z 151.386,A -85,B 0,C 180,E1 -10137.472,E2 -10137.472} C_VEL
LIN {X 0,Y 418.258,Z 151.386,A -85,B 0,C 180,E1 -10140.899,E2 -10140.899} C_VEL
LIN {X 0,Y 418.237,Z 151.515,A -85,B 0,C 180,E1 -10142.867,E2 -10142.867} C_VEL
LIN {X 0,Y 420.715,Z 163.827,A -85,B 0,C 180,E1 -10145.579,E2 -10145.579} C_VEL
LIN {X 0,Y 421.063,Z 167.665,A -85,B 0,C 180,E1 -10146.385,E2 -10146.385} C_VEL
LIN {X 0,Y 419.883,Z 186.769,A -85,B 0,C 180,E1 -10150.21,E2 -10150.21} C_VEL
LIN {X 0,Y 419.538,Z 191.315,A -85,B 0,C 180,E1 -10151.109,E2 -10151.109} C_VEL
LIN {X 0,Y 423.367,Z 216.326,A -85,B 0,C 180,E1 -10151.744,E2 -10151.744} C_VEL
LIN {X 0,Y 422.262,Z 299.282,A -85,B 0,C 180,E1 -10153.253,E2 -10153.253} C_VEL
LIN {X 0,Y 421.835,Z 312.429,A -85,B 0,C 180,E1 -10153.671,E2 -10153.671} C_VEL
LIN {X 0,Y 421.27,Z 325.151,A -85,B 0,C 180,E1 -10154.271,E2 -10154.271} C_VEL
LIN {X 0,Y 420.624,Z 336.509,A -85,B 0,C 180,E1 -10154.99,E2 -10154.99} C_VEL
LIN {X 0,Y 419.843,Z 348.238,A -85,B 0,C 180,E1 -10155.953,E2 -10155.953} C_VEL
LIN {X 0,Y 419.21,Z 358.792,A -85,B 0,C 180,E1 -10157.042,E2 -10157.042} C_VEL
LIN {X 0,Y 418.669,Z 367.422,A -85,B 0,C 180,E1 -10158.133,E2 -10158.133} C_VEL
LIN {X 0,Y 418.085,Z 375.371,A -85,B 0,C 180,E1 -10159.344,E2 -10159.344} C_VEL
LIN {X 0,Y 417.642,Z 383.122,A -85,B 0,C 180,E1 -10160.801,E2 -10160.801} C_VEL
LIN {X 0,Y 417.35,Z 389.341,A -85,B 0,C 180,E1 -10162.258,E2 -10162.258} C_VEL
LIN {X 0,Y 417.161,Z 394.273,A -85,B 0,C 180,E1 -10163.716,E2 -10163.716} C_VEL
LIN {X 0,Y 417.105,Z 398.042,A -85,B 0,C 180,E1 -10165.167,E2 -10165.167} C_VEL
LIN {X 0,Y 417.014,Z 399.984,A -85,B 0,C 180,E1 -10166.135,E2 -10166.135} C_VEL
LIN {X 0,Y 417.029,Z 401.49,A -85,B 0,C 180,E1 -10167.102,E2 -10167.102} C_VEL
LIN {X 0,Y 417.057,Z 402.538,A -85,B 0,C 180,E1 -10168.068,E2 -10168.068} C_VEL
LIN {X 0,Y 417.006,Z 403.444,A -85,B 0,C 180,E1 -10170,E2 -10170} C_VEL
LIN {X 0,Y 417.012,Z 403.286,A -85,B 0,C 180,E1 -10170.965,E2 -10170.965} C_VEL
LIN {X 0,Y 417.057,Z 402.694,A -85,B 0,C 180,E1 -10171.931,E2 -10171.931} C_VEL
LIN {X 0,Y 417.027,Z 401.706,A -85,B 0,C 180,E1 -10172.898,E2 -10172.898} C_VEL
LIN {X 0,Y 417.013,Z 400.316,A -85,B 0,C 180,E1 -10173.865,E2 -10173.865} C_VEL
LIN {X 0,Y 417.117,Z 397.386,A -85,B 0,C 180,E1 -10175.317,E2 -10175.317} C_VEL
LIN {X 0,Y 417.235,Z 393.41,A -85,B 0,C 180,E1 -10176.771,E2 -10176.771} C_VEL
LIN {X 0,Y 417.521,Z 387.304,A -85,B 0,C 180,E1 -10178.469,E2 -10178.469} C_VEL
LIN {X 0,Y 417.921,Z 380.608,A -85,B 0,C 180,E1 -10179.925,E2 -10179.925} C_VEL
LIN {X 0,Y 418.478,Z 372.3,A -85,B 0,C 180,E1 -10181.381,E2 -10181.381} C_VEL
LIN {X 0,Y 419.211,Z 363.813,A -85,B 0,C 180,E1 -10182.588,E2 -10182.588} C_VEL
LIN {X 0,Y 419.816,Z 354.043,A -85,B 0,C 180,E1 -10183.728,E2 -10183.728} C_VEL
